LIN {X 102.988,Y 84.879,Z 70.201,A 180.000,B 0.000,C 180.000} C_DIS
LIN {X 102.919,Y 84.847,Z 70.198,A 180.000,B 0.000,C 180.000} C_DIS
LIN {X 102.851,Y 84.815,Z 70.196,A 180.000,B 0.000,C 180.000} C_DIS
LIN {X 102.783,Y 84.784,Z 70.193,A 180.000,B 0.000,C 180.000} C_DIS
LIN {X 102.714,Y 84.755,Z 70.191,A 180.000,B 0.000,C 180.000} C_DIS
LIN {X 102.644,Y 84.727,Z 70.188,A 180.000,B 0.000,C 180.000} C_DIS
LIN {X 102.573,Y 84.698,Z 70.185,A 180.000,B 0.000,C 180.000} C_DIS
LIN {X 102.502,Y 84.670,Z 70.183,A 180.000,B 0.000,C 180.000} C_DIS
LIN {X 102.432,Y 84.642,Z 70.180,A 180.000,B 0.000,C 180.000} C_DIS
LIN {X 102.361,Y 84.613,Z 70.177,A 180.000,B 0.000,C 180.000} C_DIS
LIN {X 102.290,Y 84.585,Z 70.175,A 180.000,B 0.000,C 180.000} C_DIS
LIN {X 102.220,Y 84.557,Z 70.172,A 180.000,B 0.000,C 180.000} C_DIS
LIN {X 102.149,Y 84.528,Z 70.169,A 180.000,B 0.000,C 180.000} C_DIS
LIN {X 102.078,Y 84.501,Z 70.167,A 180.000,B 0.000,C 180.000} C_DIS
LIN {X 102.007,Y 84.475,Z 70.164,A 180.000,B 0.000,C 180.000} C_DIS
LIN {X 101.936,Y 84.451,Z 70.161,A 180.000,B 0.000,C 180.000} C_DIS
LIN {X 101.864,Y 84.427,Z 70.159,A 180.000,B 0.000,C 180.000} C_DIS
LIN {X 101.793,Y 84.403,Z 70.156,A 180.000,B 0.000,C 180.000} C_DIS
LIN {X 101.648,Y 84.354,Z 70.151,A 180.000,B 0.000,C 180.000} C_DIS
LIN {X 101.432,Y 84.281,Z 70.143,A 180.000,B 0.000,C 180.000} C_DIS
LIN {X 101.360,Y 84.257,Z 70.140,A 180.000,B 0.000,C 180.000} C_DIS
LIN {X 101.288,Y 84.235,Z 70.137,A 180.000,B 0.000,C 180.000} C_DIS
LIN {X 101.215,Y 84.214,Z 70.135,A 180.000,B 0.000,C 180.000} C_DIS
LIN {X 100.995,Y 84.154,Z 70.127,A 180.000,B 0.000,C 180.000} C_DIS
LIN {X 100.702,Y 84.073,Z 70.116,A 180.000,B 0.000,C 180.000} C_DIS
LIN {X 100.629,Y 84.053,Z 70.114,A 180.000,B 0.000,C 180.000} C_DIS
LIN {X 100.555,Y 84.034,Z 70.111,A 180.000,B 0.000,C 180.000} C_DIS
LIN {X 100.481,Y 84.018,Z 70.108,A 180.000,B 0.000,C 180.000} C_DIS
LIN {X 100.258,Y 83.970,Z 70.100,A 180.000,B 0.000,C 180.000} C_DIS
LIN {X 100.109,Y 83.938,Z 70.095,A 180.000,B 0.000,C 180.000} C_DIS
LIN {X 100.034,Y 83.921,Z 70.092,A 180.000,B 0.000,C 180.000} C_DIS
LIN {X 99.960,Y 83.905,Z 70.090,A 180.000,B 0.000,C 180.000} C_DIS
LIN {X 99.886,Y 83.890,Z 70.087,A 180.000,B 0.000,C 180.000} C_DIS
LIN {X 99.812,Y 83.874,Z 70.084,A 180.000,B 0.000,C 180.000} C_DIS
LIN {X 99.737,Y 83.861,Z 70.082,A 180.000,B 0.000,C 180.000} C_DIS
LIN {X 99.661,Y 83.849,Z 70.079,A 180.000,B 0.000,C 180.000} C_DIS
LIN {X 99.586,Y 83.838,Z 70.076,A 180.000,B 0.000,C 180.000} C_DIS
LIN {X 99.511,Y 83.826,Z 70.074,A 180.000,B 0.000,C 180.000} C_DIS
LIN {X 99.435,Y 83.814,Z 70.071,A 180.000,B 0.000,C 180.000} C_DIS
LIN {X 99.360,Y 83.802,Z 70.068,A 180.000,B 0.000,C 180.000} C_DIS
LIN {X 99.285,Y 83.790,Z 70.066,A 180.000,B 0.000,C 180.000} C_DIS
LIN {X 99.209,Y 83.778,Z 70.063,A 180.000,B 0.000,C 180.000} C_DIS
LIN {X 99.134,Y 83.766,Z 70.060,A 180.000,B 0.000,C 180.000} C_DIS
LIN {X 99.059,Y 83.755,Z 70.058,A 180.000,B 0.000,C 180.000} C_DIS
LIN {X 98.983,Y 83.746,Z 70.055,A 180.000,B 0.000,C 180.000} C_DIS
LIN {X 98.908,Y 83.739,Z 70.052,A 180.000,B 0.000,C 180.000} C_DIS
LIN {X 98.832,Y 83.731,Z 70.050,A 180.000,B 0.000,C 180.000} C_DIS
LIN {X 98.756,Y 83.724,Z 70.047,A 180.000,B 0.000,C 180.000} C_DIS
LIN {X 98.680,Y 83.716,Z 70.044,A 180.000,B 0.000,C 180.000} C_DIS
LIN {X 98.604,Y 83.708,Z 70.042,A 180.000,B 0.000,C 180.000} C_DIS
LIN {X 98.528,Y 83.701,Z 70.039,A 180.000,B 0.000,C 180.000} C_DIS
LIN {X 98.377,Y 83.686,Z 70.035,A 180.000,B 0.000,C 180.000} C_DIS
LIN {X 98.225,Y 83.674,Z 70.030,A 180.000,B 0.000,C 180.000} C_DIS
LIN {X 98.073,Y 83.667,Z 70.026,A 180.000,B 0.000,C 180.000} C_DIS
LIN {X 97.920,Y 83.661,Z 70.021,A 180.000,B 0.000,C 180.000} C_DIS
LIN {X 97.768,Y 83.655,Z 70.018,A 180.000,B 0.000,C 180.000} C_DIS
LIN {X 97.615,Y 83.649,Z 70.014,A 180.000,B 0.000,C 180.000} C_DIS
LIN {X 97.463,Y 83.646,Z 70.011,A 180.000,B 0.000,C 180.000} C_DIS
LIN {X 97.310,Y 83.648,Z 70.008,A 180.000,B 0.000,C 180.000} C_DIS
LIN {X 97.005,Y 83.655,Z 70.004,A 180.000,B 0.000,C 180.000} C_DIS
LIN {X 96.700,Y 83.664,Z 70.001,A 180.000,B 0.000,C 180.000} C_DIS
LIN {X 96.396,Y 83.689,Z 70.000,A 180.000,B 0.000,C 180.000} C_DIS
LIN {X 96.368,Y 83.693,Z 70.000,A 180.000,B 0.000,C 180.000} C_DIS
; Cutting Move Starts
LIN {X 96.181,Y 83.709,Z 70.000,A 180.000,B 0.000,C 180.000} C_DIS
LIN {X 96.003,Y 83.724,Z 70.000,A 180.000,B 0.000,C 180.000} C_DIS
LIN {X 95.824,Y 83.746,Z 70.000,A 180.000,B 0.000,C 180.000} C_DIS
LIN {X 95.288,Y 83.822,Z 70.000,A 180.000,B 0.000,C 180.000} C_DIS
LIN {X 95.137,Y 83.846,Z 70.000,A 180.000,B 0.000,C 180.000} C_DIS
LIN {X 95.109,Y 83.852,Z 70.000,A 180.000,B 0.000,C 180.000} C_DIS
LIN {X 94.930,Y 83.887,Z 70.000,A 180.000,B 0.000,C 180.000} C_DIS
LIN {X 94.573,Y 83.958,Z 70.000,A 180.000,B 0.000,C 180.000} C_DIS
LIN {X 94.394,Y 83.995,Z 70.000,A 180.000,B 0.000,C 180.000} C_DIS
LIN {X 94.276,Y 84.025,Z 70.000,A 180.000,B 0.000,C 180.000} C_DIS
LIN {X 93.857,Y 84.133,Z 70.000,A 180.000,B 0.000,C 180.000} C_DIS
LIN {X 93.679,Y 84.180,Z 70.000,A 180.000,B 0.000,C 180.000} C_DIS
LIN {X 93.600,Y 84.204,Z 70.000,A 180.000,B 0.000,C 180.000} C_DIS
LIN {X 93.039,Y 84.383,Z 70.000,A 180.000,B 0.000,C 180.000} C_DIS
LIN {X 92.964,Y 84.407,Z 70.000,A 180.000,B 0.000,C 180.000} C_DIS
LIN {X 92.785,Y 84.472,Z 70.000,A 180.000,B 0.000,C 180.000} C_DIS
LIN {X 92.427,Y 84.608,Z 70.000,A 180.000,B 0.000,C 180.000} C_DIS
LIN {X 92.249,Y 84.677,Z 70.000,A 180.000,B 0.000,C 180.000} C_DIS
LIN {X 92.099,Y 84.740,Z 70.000,A 180.000,B 0.000,C 180.000} C_DIS
LIN {X 91.700,Y 84.919,Z 70.000,A 180.000,B 0.000,C 180.000} C_DIS
LIN {X 91.533,Y 84.994,Z 70.000,A 180.000,B 0.000,C 180.000} C_DIS
LIN {X 91.355,Y 85.082,Z 70.000,A 180.000,B 0.000,C 180.000} C_DIS
LIN {X 90.979,Y 85.276,Z 70.000,A 180.000,B 0.000,C 180.000} C_DIS
LIN {X 90.818,Y 85.360,Z 70.000,A 180.000,B 0.000,C 180.000} C_DIS
LIN {X 90.653,Y 85.455,Z 70.000,A 180.000,B 0.000,C 180.000} C_DIS
LIN {X 90.282,Y 85.674,Z 70.000,A 180.000,B 0.000,C 180.000} C_DIS
LIN {X 90.103,Y 85.782,Z 70.000,A 180.000,B 0.000,C 180.000} C_DIS
LIN {X 90.057,Y 85.813,Z 70.000,A 180.000,B 0.000,C 180.000} C_DIS
LIN {X 89.567,Y 86.140,Z 70.000,A 180.000,B 0.000,C 180.000} C_DIS
LIN {X 89.522,Y 86.170,Z 70.000,A 180.000,B 0.000,C 180.000} C_DIS
LIN {X 89.388,Y 86.267,Z 70.000,A 180.000,B 0.000,C 180.000} C_DIS
LIN {X 89.031,Y 86.536,Z 70.000,A 180.000,B 0.000,C 180.000} C_DIS
LIN {X 88.852,Y 86.673,Z 70.000,A 180.000,B 0.000,C 180.000} C_DIS
LIN {X 88.811,Y 86.707,Z 70.000,A 180.000,B 0.000,C 180.000} C_DIS
LIN {X 88.673,Y 86.823,Z 70.000,A 180.000,B 0.000,C 180.000} C_DIS
LIN {X 88.316,Y 87.125,Z 70.000,A 180.000,B 0.000,C 180.000} C_DIS
LIN {X 88.184,Y 87.243,Z 70.000,A 180.000,B 0.000,C 180.000} C_DIS
LIN {X 87.779,Y 87.626,Z 70.000,A 180.000,B 0.000,C 180.000} C_DIS
LIN {X 87.627,Y 87.779,Z 70.000,A 180.000,B 0.000,C 180.000} C_DIS
LIN {X 87.243,Y 88.185,Z 70.000,A 180.000,B 0.000,C 180.000} C_DIS
LIN {X 87.124,Y 88.316,Z 70.000,A 180.000,B 0.000,C 180.000} C_DIS
LIN {X 87.064,Y 88.386,Z 70.000,A 180.000,B 0.000,C 180.000} C_DIS
LIN {X 86.822,Y 88.673,Z 70.000,A 180.000,B 0.000,C 180.000} C_DIS
LIN {X 86.707,Y 88.810,Z 70.000,A 180.000,B 0.000,C 180.000} C_DIS
LIN {X 86.672,Y 88.852,Z 70.000,A 180.000,B 0.000,C 180.000} C_DIS
LIN {X 86.536,Y 89.031,Z 70.000,A 180.000,B 0.000,C 180.000} C_DIS
LIN {X 86.267,Y 89.388,Z 70.000,A 180.000,B 0.000,C 180.000} C_DIS
LIN {X 86.170,Y 89.522,Z 70.000,A 180.000,B 0.000,C 180.000} C_DIS
LIN {X 86.140,Y 89.567,Z 70.000,A 180.000,B 0.000,C 180.000} C_DIS
LIN {X 85.813,Y 90.056,Z 70.000,A 180.000,B 0.000,C 180.000} C_DIS
LIN {X 85.782,Y 90.103,Z 70.000,A 180.000,B 0.000,C 180.000} C_DIS
LIN {X 85.674,Y 90.282,Z 70.000,A 180.000,B 0.000,C 180.000} C_DIS
LIN {X 85.455,Y 90.653,Z 70.000,A 180.000,B 0.000,C 180.000} C_DIS
LIN {X 85.360,Y 90.818,Z 70.000,A 180.000,B 0.000,C 180.000} C_DIS
LIN {X 85.276,Y 90.979,Z 70.000,A 180.000,B 0.000,C 180.000} C_DIS
LIN {X 85.082,Y 91.355,Z 70.000,A 180.000,B 0.000,C 180.000} C_DIS
LIN {X 84.993,Y 91.533,Z 70.000,A 180.000,B 0.000,C 180.000} C_DIS
LIN {X 84.919,Y 91.699,Z 70.000,A 180.000,B 0.000,C 180.000} C_DIS
LIN {X 84.740,Y 92.099,Z 70.000,A 180.000,B 0.000,C 180.000} C_DIS
LIN {X 84.677,Y 92.249,Z 70.000,A 180.000,B 0.000,C 180.000} C_DIS
LIN {X 84.609,Y 92.427,Z 70.000,A 180.000,B 0.000,C 180.000} C_DIS
LIN {X 84.472,Y 92.785,Z 70.000,A 180.000,B 0.000,C 180.000} C_DIS
LIN {X 84.406,Y 92.964,Z 70.000,A 180.000,B 0.000,C 180.000} C_DIS
LIN {X 84.383,Y 93.037,Z 70.000,A 180.000,B 0.000,C 180.000} C_DIS
LIN {X 84.235,Y 93.500,Z 70.000,A 180.000,B 0.000,C 180.000} C_DIS
LIN {X 84.204,Y 93.598,Z 70.000,A 180.000,B 0.000,C 180.000} C_DIS
LIN {X 84.180,Y 93.679,Z 70.000,A 180.000,B 0.000,C 180.000} C_DIS
LIN {X 84.134,Y 93.857,Z 70.000,A 180.000,B 0.000,C 180.000} C_DIS
LIN {X 84.025,Y 94.278,Z 70.000,A 180.000,B 0.000,C 180.000} C_DIS
LIN {X 83.996,Y 94.394,Z 70.000,A 180.000,B 0.000,C 180.000} C_DIS
LIN {X 83.958,Y 94.573,Z 70.000,A 180.000,B 0.000,C 180.000} C_DIS
LIN {X 83.851,Y 95.109,Z 70.000,A 180.000,B 0.000,C 180.000} C_DIS
LIN {X 83.846,Y 95.134,Z 70.000,A 180.000,B 0.000,C 180.000} C_DIS
LIN {X 83.822,Y 95.288,Z 70.000,A 180.000,B 0.000,C 180.000} C_DIS
LIN {X 83.746,Y 95.824,Z 70.000,A 180.000,B 0.000,C 180.000} C_DIS
LIN {X 83.724,Y 96.003,Z 70.000,A 180.000,B 0.000,C 180.000} C_DIS
LIN {X 83.709,Y 96.181,Z 70.000,A 180.000,B 0.000,C 180.000} C_DIS
LIN {X 83.679,Y 96.539,Z 70.000,A 180.000,B 0.000,C 180.000} C_DIS
LIN {X 83.668,Y 96.673,Z 70.000,A 180.000,B 0.000,C 180.000} C_DIS
LIN {X 83.665,Y 96.718,Z 70.000,A 180.000,B 0.000,C 180.000} C_DIS
LIN {X 83.659,Y 96.897,Z 70.000,A 180.000,B 0.000,C 180.000} C_DIS
LIN {X 83.648,Y 97.254,Z 70.000,A 180.000,B 0.000,C 180.000} C_DIS
LIN {X 83.644,Y 97.433,Z 70.000,A 180.000,B 0.000,C 180.000} C_DIS
LIN {X 83.645,Y 97.612,Z 70.000,A 180.000,B 0.000,C 180.000} C_DIS
LIN {X 83.660,Y 98.148,Z 70.000,A 180.000,B 0.000,C 180.000} C_DIS
LIN {X 83.668,Y 98.327,Z 70.000,A 180.000,B 0.000,C 180.000} C_DIS
LIN {X 83.683,Y 98.505,Z 70.000,A 180.000,B 0.000,C 180.000} C_DIS
LIN {X 83.713,Y 98.863,Z 70.000,A 180.000,B 0.000,C 180.000} C_DIS
LIN {X 83.729,Y 99.042,Z 70.000,A 180.000,B 0.000,C 180.000} C_DIS
LIN {X 83.753,Y 99.221,Z 70.000,A 180.000,B 0.000,C 180.000} C_DIS
LIN {X 83.828,Y 99.757,Z 70.000,A 180.000,B 0.000,C 180.000} C_DIS
LIN {X 83.846,Y 99.866,Z 70.000,A 180.000,B 0.000,C 180.000} C_DIS
LIN {X 83.860,Y 99.936,Z 70.000,A 180.000,B 0.000,C 180.000} C_DIS
LIN {X 83.967,Y 100.472,Z 70.000,A 180.000,B 0.000,C 180.000} C_DIS
LIN {X 84.007,Y 100.651,Z 70.000,A 180.000,B 0.000,C 180.000} C_DIS
LIN {X 84.025,Y 100.722,Z 70.000,A 180.000,B 0.000,C 180.000} C_DIS
LIN {X 84.145,Y 101.187,Z 70.000,A 180.000,B 0.000,C 180.000} C_DIS
LIN {X 84.193,Y 101.366,Z 70.000,A 180.000,B 0.000,C 180.000} C_DIS
LIN {X 84.204,Y 101.402,Z 70.000,A 180.000,B 0.000,C 180.000} C_DIS
LIN {X 84.249,Y 101.545,Z 70.000,A 180.000,B 0.000,C 180.000} C_DIS
LIN {X 84.383,Y 101.963,Z 70.000,A 180.000,B 0.000,C 180.000} C_DIS
LIN {X 84.422,Y 102.081,Z 70.000,A 180.000,B 0.000,C 180.000} C_DIS
LIN {X 84.489,Y 102.260,Z 70.000,A 180.000,B 0.000,C 180.000} C_DIS
LIN {X 84.626,Y 102.617,Z 70.000,A 180.000,B 0.000,C 180.000} C_DIS
LIN {X 84.695,Y 102.796,Z 70.000,A 180.000,B 0.000,C 180.000} C_DIS
LIN {X 84.740,Y 102.901,Z 70.000,A 180.000,B 0.000,C 180.000} C_DIS
LIN {X 84.933,Y 103.332,Z 70.000,A 180.000,B 0.000,C 180.000} C_DIS
LIN {X 85.014,Y 103.511,Z 70.000,A 180.000,B 0.000,C 180.000} C_DIS
LIN {X 85.098,Y 103.675,Z 70.000,A 180.000,B 0.000,C 180.000} C_DIS
LIN {X 85.290,Y 104.047,Z 70.000,A 180.000,B 0.000,C 180.000} C_DIS
LIN {X 85.385,Y 104.226,Z 70.000,A 180.000,B 0.000,C 180.000} C_DIS
LIN {X 85.455,Y 104.347,Z 70.000,A 180.000,B 0.000,C 180.000} C_DIS
LIN {X 85.700,Y 104.762,Z 70.000,A 180.000,B 0.000,C 180.000} C_DIS
LIN {X 85.811,Y 104.941,Z 70.000,A 180.000,B 0.000,C 180.000} C_DIS
LIN {X 86.050,Y 105.299,Z 70.000,A 180.000,B 0.000,C 180.000} C_DIS
LIN {X 86.170,Y 105.477,Z 70.000,A 180.000,B 0.000,C 180.000} C_DIS
LIN {X 86.170,Y 105.478,Z 70.000,A 180.000,B 0.000,C 180.000} C_DIS
LIN {X 86.301,Y 105.656,Z 70.000,A 180.000,B 0.000,C 180.000} C_DIS
LIN {X 86.570,Y 106.014,Z 70.000,A 180.000,B 0.000,C 180.000} C_DIS
LIN {X 86.707,Y 106.190,Z 70.000,A 180.000,B 0.000,C 180.000} C_DIS
LIN {X 86.709,Y 106.193,Z 70.000,A 180.000,B 0.000,C 180.000} C_DIS
LIN {X 86.885,Y 106.402,Z 70.000,A 180.000,B 0.000,C 180.000} C_DIS
LIN {X 87.064,Y 106.614,Z 70.000,A 180.000,B 0.000,C 180.000} C_DIS
LIN {X 87.163,Y 106.729,Z 70.000,A 180.000,B 0.000,C 180.000} C_DIS
LIN {X 87.243,Y 106.815,Z 70.000,A 180.000,B 0.000,C 180.000} C_DIS
LIN {X 87.601,Y 107.193,Z 70.000,A 180.000,B 0.000,C 180.000} C_DIS
LIN {X 87.669,Y 107.265,Z 70.000,A 180.000,B 0.000,C 180.000} C_DIS
LIN {X 87.779,Y 107.374,Z 70.000,A 180.000,B 0.000,C 180.000} C_DIS
LIN {X 88.137,Y 107.712,Z 70.000,A 180.000,B 0.000,C 180.000} C_DIS
LIN {X 88.232,Y 107.802,Z 70.000,A 180.000,B 0.000,C 180.000} C_DIS
LIN {X 88.316,Y 107.875,Z 70.000,A 180.000,B 0.000,C 180.000} C_DIS
LIN {X 88.673,Y 108.177,Z 70.000,A 180.000,B 0.000,C 180.000} C_DIS
LIN {X 88.852,Y 108.327,Z 70.000,A 180.000,B 0.000,C 180.000} C_DIS
LIN {X 88.865,Y 108.338,Z 70.000,A 180.000,B 0.000,C 180.000} C_DIS
LIN {X 89.031,Y 108.464,Z 70.000,A 180.000,B 0.000,C 180.000} C_DIS
LIN {X 89.388,Y 108.733,Z 70.000,A 180.000,B 0.000,C 180.000} C_DIS
LIN {X 89.567,Y 108.860,Z 70.000,A 180.000,B 0.000,C 180.000} C_DIS
LIN {X 89.925,Y 109.099,Z 70.000,A 180.000,B 0.000,C 180.000} C_DIS
LIN {X 90.103,Y 109.218,Z 70.000,A 180.000,B 0.000,C 180.000} C_DIS
LIN {X 90.125,Y 109.232,Z 70.000,A 180.000,B 0.000,C 180.000} C_DIS
LIN {X 90.282,Y 109.326,Z 70.000,A 180.000,B 0.000,C 180.000} C_DIS
LIN {X 90.728,Y 109.589,Z 70.000,A 180.000,B 0.000,C 180.000} C_DIS
LIN {X 90.818,Y 109.640,Z 70.000,A 180.000,B 0.000,C 180.000} C_DIS
LIN {X 90.997,Y 109.733,Z 70.000,A 180.000,B 0.000,C 180.000} C_DIS
LIN {X 91.411,Y 109.947,Z 70.000,A 180.000,B 0.000,C 180.000} C_DIS
LIN {X 91.533,Y 110.006,Z 70.000,A 180.000,B 0.000,C 180.000} C_DIS
LIN {X 91.712,Y 110.087,Z 70.000,A 180.000,B 0.000,C 180.000} C_DIS
LIN {X 92.070,Y 110.247,Z 70.000,A 180.000,B 0.000,C 180.000} C_DIS
LIN {X 92.201,Y 110.304,Z 70.000,A 180.000,B 0.000,C 180.000} C_DIS
LIN {X 92.249,Y 110.323,Z 70.000,A 180.000,B 0.000,C 180.000} C_DIS
LIN {X 92.427,Y 110.392,Z 70.000,A 180.000,B 0.000,C 180.000} C_DIS
LIN {X 92.785,Y 110.528,Z 70.000,A 180.000,B 0.000,C 180.000} C_DIS
LIN {X 92.964,Y 110.593,Z 70.000,A 180.000,B 0.000,C 180.000} C_DIS
LIN {X 93.142,Y 110.650,Z 70.000,A 180.000,B 0.000,C 180.000} C_DIS
LIN {X 93.500,Y 110.764,Z 70.000,A 180.000,B 0.000,C 180.000} C_DIS
LIN {X 93.679,Y 110.820,Z 70.000,A 180.000,B 0.000,C 180.000} C_DIS
LIN {X 93.755,Y 110.841,Z 70.000,A 180.000,B 0.000,C 180.000} C_DIS
LIN {X 94.215,Y 110.959,Z 70.000,A 180.000,B 0.000,C 180.000} C_DIS
LIN {X 94.394,Y 111.005,Z 70.000,A 180.000,B 0.000,C 180.000} C_DIS
LIN {X 94.460,Y 111.019,Z 70.000,A 180.000,B 0.000,C 180.000} C_DIS
LIN {X 94.573,Y 111.042,Z 70.000,A 180.000,B 0.000,C 180.000} C_DIS
LIN {X 94.930,Y 111.113,Z 70.000,A 180.000,B 0.000,C 180.000} C_DIS
LIN {X 95.109,Y 111.148,Z 70.000,A 180.000,B 0.000,C 180.000} C_DIS
LIN {X 95.288,Y 111.178,Z 70.000,A 180.000,B 0.000,C 180.000} C_DIS
LIN {X 95.824,Y 111.254,Z 70.000,A 180.000,B 0.000,C 180.000} C_DIS
LIN {X 96.003,Y 111.276,Z 70.000,A 180.000,B 0.000,C 180.000} C_DIS
LIN {X 96.181,Y 111.291,Z 70.000,A 180.000,B 0.000,C 180.000} C_DIS
LIN {X 96.539,Y 111.321,Z 70.000,A 180.000,B 0.000,C 180.000} C_DIS
LIN {X 96.718,Y 111.335,Z 70.000,A 180.000,B 0.000,C 180.000} C_DIS
LIN {X 96.897,Y 111.342,Z 70.000,A 180.000,B 0.000,C 180.000} C_DIS
LIN {X 97.433,Y 111.357,Z 70.000,A 180.000,B 0.000,C 180.000} C_DIS
LIN {X 97.612,Y 111.355,Z 70.000,A 180.000,B 0.000,C 180.000} C_DIS
LIN {X 98.148,Y 111.340,Z 70.000,A 180.000,B 0.000,C 180.000} C_DIS
LIN {X 98.327,Y 111.332,Z 70.000,A 180.000,B 0.000,C 180.000} C_DIS
LIN {X 98.505,Y 111.317,Z 70.000,A 180.000,B 0.000,C 180.000} C_DIS
LIN {X 98.863,Y 111.287,Z 70.000,A 180.000,B 0.000,C 180.000} C_DIS
LIN {X 99.042,Y 111.271,Z 70.000,A 180.000,B 0.000,C 180.000} C_DIS
LIN {X 99.221,Y 111.248,Z 70.000,A 180.000,B 0.000,C 180.000} C_DIS
LIN {X 99.578,Y 111.197,Z 70.000,A 180.000,B 0.000,C 180.000} C_DIS
LIN {X 99.757,Y 111.172,Z 70.000,A 180.000,B 0.000,C 180.000} C_DIS
LIN {X 99.936,Y 111.140,Z 70.000,A 180.000,B 0.000,C 180.000} C_DIS
LIN {X 100.472,Y 111.033,Z 70.000,A 180.000,B 0.000,C 180.000} C_DIS
LIN {X 100.540,Y 111.019,Z 70.000,A 180.000,B 0.000,C 180.000} C_DIS
LIN {X 100.651,Y 110.994,Z 70.000,A 180.000,B 0.000,C 180.000} C_DIS
LIN {X 100.829,Y 110.948,Z 70.000,A 180.000,B 0.000,C 180.000} C_DIS
LIN {X 101.245,Y 110.841,Z 70.000,A 180.000,B 0.000,C 180.000} C_DIS
LIN {X 101.366,Y 110.807,Z 70.000,A 180.000,B 0.000,C 180.000} C_DIS
LIN {X 101.545,Y 110.750,Z 70.000,A 180.000,B 0.000,C 180.000} C_DIS
LIN {X 101.902,Y 110.636,Z 70.000,A 180.000,B 0.000,C 180.000} C_DIS
LIN {X 102.081,Y 110.578,Z 70.000,A 180.000,B 0.000,C 180.000} C_DIS
LIN {X 102.260,Y 110.511,Z 70.000,A 180.000,B 0.000,C 180.000} C_DIS
LIN {X 102.617,Y 110.375,Z 70.000,A 180.000,B 0.000,C 180.000} C_DIS
LIN {X 102.796,Y 110.306,Z 70.000,A 180.000,B 0.000,C 180.000} C_DIS
LIN {X 102.799,Y 110.304,Z 70.000,A 180.000,B 0.000,C 180.000} C_DIS
LIN {X 102.975,Y 110.227,Z 70.000,A 180.000,B 0.000,C 180.000} C_DIS
LIN {X 103.332,Y 110.067,Z 70.000,A 180.000,B 0.000,C 180.000} C_DIS
LIN {X 103.511,Y 109.985,Z 70.000,A 180.000,B 0.000,C 180.000} C_DIS
LIN {X 103.589,Y 109.947,Z 70.000,A 180.000,B 0.000,C 180.000} C_DIS
LIN {X 104.047,Y 109.710,Z 70.000,A 180.000,B 0.000,C 180.000} C_DIS
LIN {X 104.226,Y 109.616,Z 70.000,A 180.000,B 0.000,C 180.000} C_DIS
LIN {X 104.272,Y 109.589,Z 70.000,A 180.000,B 0.000,C 180.000} C_DIS
LIN {X 104.762,Y 109.300,Z 70.000,A 180.000,B 0.000,C 180.000} C_DIS
LIN {X 104.875,Y 109.232,Z 70.000,A 180.000,B 0.000,C 180.000} C_DIS
LIN {X 104.941,Y 109.189,Z 70.000,A 180.000,B 0.000,C 180.000} C_DIS
LIN {X 105.145,Y 109.053,Z 70.000,A 180.000,B 0.000,C 180.000} C_DIS
LIN {X 105.412,Y 108.874,Z 70.000,A 180.000,B 0.000,C 180.000} C_DIS
LIN {X 105.477,Y 108.830,Z 70.000,A 180.000,B 0.000,C 180.000} C_DIS
LIN {X 105.656,Y 108.700,Z 70.000,A 180.000,B 0.000,C 180.000} C_DIS
LIN {X 106.014,Y 108.431,Z 70.000,A 180.000,B 0.000,C 180.000} C_DIS
LIN {X 106.135,Y 108.338,Z 70.000,A 180.000,B 0.000,C 180.000} C_DIS
LIN {X 106.193,Y 108.291,Z 70.000,A 180.000,B 0.000,C 180.000} C_DIS
LIN {X 106.349,Y 108.159,Z 70.000,A 180.000,B 0.000,C 180.000} C_DIS
LIN {X 106.560,Y 107.980,Z 70.000,A 180.000,B 0.000,C 180.000} C_DIS
LIN {X 106.729,Y 107.837,Z 70.000,A 180.000,B 0.000,C 180.000} C_DIS
LIN {X 106.768,Y 107.802,Z 70.000,A 180.000,B 0.000,C 180.000} C_DIS
LIN {X 106.908,Y 107.670,Z 70.000,A 180.000,B 0.000,C 180.000} C_DIS
LIN {X 107.147,Y 107.444,Z 70.000,A 180.000,B 0.000,C 180.000} C_DIS
LIN {X 107.265,Y 107.332,Z 70.000,A 180.000,B 0.000,C 180.000} C_DIS
LIN {X 107.331,Y 107.265,Z 70.000,A 180.000,B 0.000,C 180.000} C_DIS
LIN {X 107.444,Y 107.146,Z 70.000,A 180.000,B 0.000,C 180.000} C_DIS
LIN {X 107.669,Y 106.908,Z 70.000,A 180.000,B 0.000,C 180.000} C_DIS
LIN {X 107.802,Y 106.768,Z 70.000,A 180.000,B 0.000,C 180.000} C_DIS
LIN {X 107.837,Y 106.729,Z 70.000,A 180.000,B 0.000,C 180.000} C_DIS
LIN {X 107.980,Y 106.561,Z 70.000,A 180.000,B 0.000,C 180.000} C_DIS
LIN {X 108.159,Y 106.349,Z 70.000,A 180.000,B 0.000,C 180.000} C_DIS
LIN {X 108.291,Y 106.193,Z 70.000,A 180.000,B 0.000,C 180.000} C_DIS
LIN {X 108.338,Y 106.135,Z 70.000,A 180.000,B 0.000,C 180.000} C_DIS
LIN {X 108.430,Y 106.014,Z 70.000,A 180.000,B 0.000,C 180.000} C_DIS
LIN {X 108.699,Y 105.656,Z 70.000,A 180.000,B 0.000,C 180.000} C_DIS
LIN {X 108.830,Y 105.477,Z 70.000,A 180.000,B 0.000,C 180.000} C_DIS
LIN {X 108.874,Y 105.412,Z 70.000,A 180.000,B 0.000,C 180.000} C_DIS
LIN {X 109.189,Y 104.941,Z 70.000,A 180.000,B 0.000,C 180.000} C_DIS
LIN {X 109.232,Y 104.876,Z 70.000,A 180.000,B 0.000,C 180.000} C_DIS
LIN {X 109.300,Y 104.762,Z 70.000,A 180.000,B 0.000,C 180.000} C_DIS
LIN {X 109.511,Y 104.405,Z 70.000,A 180.000,B 0.000,C 180.000} C_DIS
LIN {X 109.589,Y 104.271,Z 70.000,A 180.000,B 0.000,C 180.000} C_DIS
LIN {X 109.615,Y 104.226,Z 70.000,A 180.000,B 0.000,C 180.000} C_DIS
LIN {X 109.710,Y 104.047,Z 70.000,A 180.000,B 0.000,C 180.000} C_DIS
LIN {X 109.947,Y 103.589,Z 70.000,A 180.000,B 0.000,C 180.000} C_DIS
LIN {X 109.986,Y 103.511,Z 70.000,A 180.000,B 0.000,C 180.000} C_DIS
LIN {X 110.067,Y 103.332,Z 70.000,A 180.000,B 0.000,C 180.000} C_DIS
LIN {X 110.227,Y 102.975,Z 70.000,A 180.000,B 0.000,C 180.000} C_DIS
LIN {X 110.304,Y 102.798,Z 70.000,A 180.000,B 0.000,C 180.000} C_DIS
LIN {X 110.305,Y 102.796,Z 70.000,A 180.000,B 0.000,C 180.000} C_DIS
LIN {X 110.374,Y 102.617,Z 70.000,A 180.000,B 0.000,C 180.000} C_DIS
LIN {X 110.511,Y 102.260,Z 70.000,A 180.000,B 0.000,C 180.000} C_DIS
LIN {X 110.578,Y 102.081,Z 70.000,A 180.000,B 0.000,C 180.000} C_DIS
LIN {X 110.637,Y 101.902,Z 70.000,A 180.000,B 0.000,C 180.000} C_DIS
LIN {X 110.751,Y 101.545,Z 70.000,A 180.000,B 0.000,C 180.000} C_DIS
LIN {X 110.807,Y 101.366,Z 70.000,A 180.000,B 0.000,C 180.000} C_DIS
LIN {X 110.841,Y 101.243,Z 70.000,A 180.000,B 0.000,C 180.000} C_DIS
LIN {X 110.947,Y 100.829,Z 70.000,A 180.000,B 0.000,C 180.000} C_DIS
LIN {X 110.993,Y 100.651,Z 70.000,A 180.000,B 0.000,C 180.000} C_DIS
LIN {X 111.019,Y 100.541,Z 70.000,A 180.000,B 0.000,C 180.000} C_DIS
LIN {X 111.033,Y 100.472,Z 70.000,A 180.000,B 0.000,C 180.000} C_DIS
LIN {X 111.140,Y 99.936,Z 70.000,A 180.000,B 0.000,C 180.000} C_DIS
LIN {X 111.172,Y 99.757,Z 70.000,A 180.000,B 0.000,C 180.000} C_DIS
LIN {X 111.247,Y 99.221,Z 70.000,A 180.000,B 0.000,C 180.000} C_DIS
LIN {X 111.271,Y 99.042,Z 70.000,A 180.000,B 0.000,C 180.000} C_DIS
LIN {X 111.287,Y 98.863,Z 70.000,A 180.000,B 0.000,C 180.000} C_DIS
LIN {X 111.317,Y 98.505,Z 70.000,A 180.000,B 0.000,C 180.000} C_DIS
LIN {X 111.332,Y 98.327,Z 70.000,A 180.000,B 0.000,C 180.000} C_DIS
LIN {X 111.340,Y 98.148,Z 70.000,A 180.000,B 0.000,C 180.000} C_DIS
LIN {X 111.355,Y 97.612,Z 70.000,A 180.000,B 0.000,C 180.000} C_DIS
LIN {X 111.356,Y 97.433,Z 70.000,A 180.000,B 0.000,C 180.000} C_DIS
LIN {X 111.352,Y 97.254,Z 70.000,A 180.000,B 0.000,C 180.000} C_DIS
LIN {X 111.341,Y 96.897,Z 70.000,A 180.000,B 0.000,C 180.000} C_DIS
LIN {X 111.335,Y 96.718,Z 70.000,A 180.000,B 0.000,C 180.000} C_DIS
LIN {X 111.321,Y 96.539,Z 70.000,A 180.000,B 0.000,C 180.000} C_DIS
LIN {X 111.291,Y 96.181,Z 70.000,A 180.000,B 0.000,C 180.000} C_DIS
LIN {X 111.276,Y 96.003,Z 70.000,A 180.000,B 0.000,C 180.000} C_DIS
LIN {X 111.254,Y 95.824,Z 70.000,A 180.000,B 0.000,C 180.000} C_DIS
LIN {X 111.178,Y 95.288,Z 70.000,A 180.000,B 0.000,C 180.000} C_DIS
LIN {X 111.149,Y 95.109,Z 70.000,A 180.000,B 0.000,C 180.000} C_DIS
LIN {X 111.042,Y 94.573,Z 70.000,A 180.000,B 0.000,C 180.000} C_DIS
LIN {X 111.019,Y 94.459,Z 70.000,A 180.000,B 0.000,C 180.000} C_DIS
LIN {X 111.004,Y 94.394,Z 70.000,A 180.000,B 0.000,C 180.000} C_DIS
LIN {X 110.959,Y 94.215,Z 70.000,A 180.000,B 0.000,C 180.000} C_DIS
LIN {X 110.841,Y 93.757,Z 70.000,A 180.000,B 0.000,C 180.000} C_DIS
LIN {X 110.820,Y 93.679,Z 70.000,A 180.000,B 0.000,C 180.000} C_DIS
LIN {X 110.765,Y 93.500,Z 70.000,A 180.000,B 0.000,C 180.000} C_DIS
LIN {X 110.651,Y 93.142,Z 70.000,A 180.000,B 0.000,C 180.000} C_DIS
LIN {X 110.594,Y 92.964,Z 70.000,A 180.000,B 0.000,C 180.000} C_DIS
LIN {X 110.528,Y 92.785,Z 70.000,A 180.000,B 0.000,C 180.000} C_DIS
LIN {X 110.391,Y 92.427,Z 70.000,A 180.000,B 0.000,C 180.000} C_DIS
LIN {X 110.323,Y 92.249,Z 70.000,A 180.000,B 0.000,C 180.000} C_DIS
LIN {X 110.304,Y 92.202,Z 70.000,A 180.000,B 0.000,C 180.000} C_DIS
LIN {X 110.247,Y 92.070,Z 70.000,A 180.000,B 0.000,C 180.000} C_DIS
LIN {X 110.087,Y 91.712,Z 70.000,A 180.000,B 0.000,C 180.000} C_DIS
LIN {X 110.007,Y 91.533,Z 70.000,A 180.000,B 0.000,C 180.000} C_DIS
LIN {X 109.947,Y 91.411,Z 70.000,A 180.000,B 0.000,C 180.000} C_DIS
LIN {X 109.733,Y 90.997,Z 70.000,A 180.000,B 0.000,C 180.000} C_DIS
LIN {X 109.640,Y 90.818,Z 70.000,A 180.000,B 0.000,C 180.000} C_DIS
LIN {X 109.589,Y 90.729,Z 70.000,A 180.000,B 0.000,C 180.000} C_DIS
LIN {X 109.537,Y 90.640,Z 70.000,A 180.000,B 0.000,C 180.000} C_DIS
LIN {X 109.326,Y 90.282,Z 70.000,A 180.000,B 0.000,C 180.000} C_DIS
LIN {X 109.232,Y 90.124,Z 70.000,A 180.000,B 0.000,C 180.000} C_DIS
LIN {X 109.218,Y 90.103,Z 70.000,A 180.000,B 0.000,C 180.000} C_DIS
LIN {X 109.099,Y 89.925,Z 70.000,A 180.000,B 0.000,C 180.000} C_DIS
LIN {X 108.860,Y 89.567,Z 70.000,A 180.000,B 0.000,C 180.000} C_DIS
LIN {X 108.733,Y 89.388,Z 70.000,A 180.000,B 0.000,C 180.000} C_DIS
LIN {X 108.464,Y 89.031,Z 70.000,A 180.000,B 0.000,C 180.000} C_DIS
LIN {X 108.338,Y 88.865,Z 70.000,A 180.000,B 0.000,C 180.000} C_DIS
LIN {X 108.328,Y 88.852,Z 70.000,A 180.000,B 0.000,C 180.000} C_DIS
LIN {X 108.178,Y 88.673,Z 70.000,A 180.000,B 0.000,C 180.000} C_DIS
LIN {X 107.980,Y 88.439,Z 70.000,A 180.000,B 0.000,C 180.000} C_DIS
LIN {X 107.876,Y 88.316,Z 70.000,A 180.000,B 0.000,C 180.000} C_DIS
LIN {X 107.802,Y 88.232,Z 70.000,A 180.000,B 0.000,C 180.000} C_DIS
LIN {X 107.711,Y 88.137,Z 70.000,A 180.000,B 0.000,C 180.000} C_DIS
LIN {X 107.373,Y 87.779,Z 70.000,A 180.000,B 0.000,C 180.000} C_DIS
LIN {X 107.265,Y 87.668,Z 70.000,A 180.000,B 0.000,C 180.000} C_DIS
LIN {X 107.194,Y 87.601,Z 70.000,A 180.000,B 0.000,C 180.000} C_DIS
LIN {X 106.816,Y 87.243,Z 70.000,A 180.000,B 0.000,C 180.000} C_DIS
LIN {X 106.729,Y 87.163,Z 70.000,A 180.000,B 0.000,C 180.000} C_DIS
LIN {X 106.613,Y 87.064,Z 70.000,A 180.000,B 0.000,C 180.000} C_DIS
LIN {X 106.371,Y 86.860,Z 70.000,A 180.000,B 0.000,C 180.000} C_DIS
LIN {X 106.193,Y 86.709,Z 70.000,A 180.000,B 0.000,C 180.000} C_DIS
LIN {X 106.189,Y 86.707,Z 70.000,A 180.000,B 0.000,C 180.000} C_DIS
LIN {X 106.014,Y 86.569,Z 70.000,A 180.000,B 0.000,C 180.000} C_DIS
LIN {X 105.656,Y 86.300,Z 70.000,A 180.000,B 0.000,C 180.000} C_DIS
LIN {X 105.478,Y 86.170,Z 70.000,A 180.000,B 0.000,C 180.000} C_DIS
LIN {X 105.477,Y 86.170,Z 70.000,A 180.000,B 0.000,C 180.000} C_DIS
LIN {X 105.299,Y 86.050,Z 70.000,A 180.000,B 0.000,C 180.000} C_DIS
LIN {X 105.103,Y 85.920,Z 70.000,A 180.000,B 0.000,C 180.000} C_DIS
LIN {X 104.943,Y 85.813,Z 70.000,A 180.000,B 0.000,C 180.000} C_DIS
LIN {X 104.941,Y 85.811,Z 70.000,A 180.000,B 0.000,C 180.000} C_DIS
LIN {X 104.762,Y 85.700,Z 70.000,A 180.000,B 0.000,C 180.000} C_DIS
LIN {X 104.347,Y 85.455,Z 70.000,A 180.000,B 0.000,C 180.000} C_DIS
LIN {X 104.226,Y 85.384,Z 70.000,A 180.000,B 0.000,C 180.000} C_DIS
LIN {X 104.047,Y 85.290,Z 70.000,A 180.000,B 0.000,C 180.000} C_DIS
LIN {X 103.675,Y 85.098,Z 70.000,A 180.000,B 0.000,C 180.000} C_DIS
LIN {X 103.511,Y 85.015,Z 70.000,A 180.000,B 0.000,C 180.000} C_DIS
LIN {X 103.332,Y 84.933,Z 70.000,A 180.000,B 0.000,C 180.000} C_DIS
LIN {X 102.901,Y 84.740,Z 70.000,A 180.000,B 0.000,C 180.000} C_DIS
LIN {X 102.796,Y 84.694,Z 70.000,A 180.000,B 0.000,C 180.000} C_DIS
LIN {X 102.617,Y 84.625,Z 70.000,A 180.000,B 0.000,C 180.000} C_DIS
LIN {X 102.260,Y 84.489,Z 70.000,A 180.000,B 0.000,C 180.000} C_DIS
LIN {X 102.081,Y 84.422,Z 70.000,A 180.000,B 0.000,C 180.000} C_DIS
LIN {X 101.961,Y 84.383,Z 70.000,A 180.000,B 0.000,C 180.000} C_DIS
LIN {X 101.400,Y 84.204,Z 70.000,A 180.000,B 0.000,C 180.000} C_DIS
LIN {X 101.366,Y 84.193,Z 70.000,A 180.000,B 0.000,C 180.000} C_DIS
LIN {X 101.187,Y 84.144,Z 70.000,A 180.000,B 0.000,C 180.000} C_DIS
LIN {X 100.724,Y 84.025,Z 70.000,A 180.000,B 0.000,C 180.000} C_DIS
LIN {X 100.651,Y 84.006,Z 70.000,A 180.000,B 0.000,C 180.000} C_DIS
LIN {X 100.472,Y 83.967,Z 70.000,A 180.000,B 0.000,C 180.000} C_DIS
LIN {X 99.936,Y 83.860,Z 70.000,A 180.000,B 0.000,C 180.000} C_DIS
LIN {X 99.863,Y 83.846,Z 70.000,A 180.000,B 0.000,C 180.000} C_DIS
LIN {X 99.757,Y 83.828,Z 70.000,A 180.000,B 0.000,C 180.000} C_DIS
LIN {X 99.578,Y 83.803,Z 70.000,A 180.000,B 0.000,C 180.000} C_DIS
LIN {X 99.221,Y 83.752,Z 70.000,A 180.000,B 0.000,C 180.000} C_DIS
LIN {X 99.042,Y 83.729,Z 70.000,A 180.000,B 0.000,C 180.000} C_DIS
LIN {X 98.863,Y 83.713,Z 70.000,A 180.000,B 0.000,C 180.000} C_DIS
LIN {X 98.505,Y 83.683,Z 70.000,A 180.000,B 0.000,C 180.000} C_DIS
LIN {X 98.327,Y 83.668,Z 70.000,A 180.000,B 0.000,C 180.000} C_DIS
LIN {X 98.321,Y 83.668,Z 70.000,A 180.000,B 0.000,C 180.000} C_DIS
LIN {X 98.148,Y 83.660,Z 70.000,A 180.000,B 0.000,C 180.000} C_DIS
LIN {X 97.612,Y 83.645,Z 70.000,A 180.000,B 0.000,C 180.000} C_DIS
LIN {X 97.433,Y 83.643,Z 70.000,A 180.000,B 0.000,C 180.000} C_DIS
LIN {X 96.897,Y 83.658,Z 70.000,A 180.000,B 0.000,C 180.000} C_DIS
LIN {X 96.718,Y 83.665,Z 70.000,A 180.000,B 0.000,C 180.000} C_DIS
LIN {X 96.679,Y 83.668,Z 70.000,A 180.000,B 0.000,C 180.000} C_DIS
LIN {X 96.539,Y 83.679,Z 70.000,A 180.000,B 0.000,C 180.000} C_DIS
LIN {X 96.368,Y 83.693,Z 70.000,A 180.000,B 0.000,C 180.000} C_DIS
; Link Move Starts
LIN {X 96.054,Y 83.717,Z 70.000,A 180.000,B 0.000,C 180.000} C_DIS
LIN {X 95.767,Y 83.751,Z 69.999,A 180.000,B 0.000,C 180.000} C_DIS
LIN {X 95.455,Y 83.795,Z 69.998,A 180.000,B 0.000,C 180.000} C_DIS
LIN {X 95.166,Y 83.837,Z 69.996,A 180.000,B 0.000,C 180.000} C_DIS
LIN {X 94.860,Y 83.896,Z 69.994,A 180.000,B 0.000,C 180.000} C_DIS
LIN {X 94.551,Y 83.956,Z 69.992,A 180.000,B 0.000,C 180.000} C_DIS
LIN {X 94.269,Y 84.019,Z 69.989,A 180.000,B 0.000,C 180.000} C_DIS
LIN {X 93.963,Y 84.096,Z 69.986,A 180.000,B 0.000,C 180.000} C_DIS
LIN {X 93.664,Y 84.173,Z 69.982,A 180.000,B 0.000,C 180.000} C_DIS
LIN {X 93.382,Y 84.260,Z 69.978,A 180.000,B 0.000,C 180.000} C_DIS
LIN {X 93.082,Y 84.353,Z 69.974,A 180.000,B 0.000,C 180.000} C_DIS
LIN {X 92.801,Y 84.447,Z 69.969,A 180.000,B 0.000,C 180.000} C_DIS
LIN {X 92.656,Y 84.502,Z 69.966,A 180.000,B 0.000,C 180.000} C_DIS
LIN {X 92.511,Y 84.556,Z 69.964,A 180.000,B 0.000,C 180.000} C_DIS
LIN {X 92.372,Y 84.607,Z 69.961,A 180.000,B 0.000,C 180.000} C_DIS
LIN {X 92.233,Y 84.659,Z 69.958,A 180.000,B 0.000,C 180.000} C_DIS
LIN {X 92.091,Y 84.719,Z 69.955,A 180.000,B 0.000,C 180.000} C_DIS
LIN {X 91.950,Y 84.780,Z 69.952,A 180.000,B 0.000,C 180.000} C_DIS
LIN {X 91.805,Y 84.843,Z 69.949,A 180.000,B 0.000,C 180.000} C_DIS
LIN {X 91.661,Y 84.906,Z 69.946,A 180.000,B 0.000,C 180.000} C_DIS
LIN {X 91.523,Y 84.966,Z 69.943,A 180.000,B 0.000,C 180.000} C_DIS
LIN {X 91.388,Y 85.031,Z 69.939,A 180.000,B 0.000,C 180.000} C_DIS
LIN {X 91.252,Y 85.099,Z 69.936,A 180.000,B 0.000,C 180.000} C_DIS
LIN {X 91.115,Y 85.168,Z 69.932,A 180.000,B 0.000,C 180.000} C_DIS
LIN {X 90.980,Y 85.236,Z 69.929,A 180.000,B 0.000,C 180.000} C_DIS
LIN {X 90.844,Y 85.304,Z 69.925,A 180.000,B 0.000,C 180.000} C_DIS
LIN {X 90.711,Y 85.376,Z 69.922,A 180.000,B 0.000,C 180.000} C_DIS
LIN {X 90.580,Y 85.451,Z 69.918,A 180.000,B 0.000,C 180.000} C_DIS
LIN {X 90.443,Y 85.530,Z 69.914,A 180.000,B 0.000,C 180.000} C_DIS
LIN {X 90.307,Y 85.608,Z 69.910,A 180.000,B 0.000,C 180.000} C_DIS
LIN {X 90.177,Y 85.682,Z 69.906,A 180.000,B 0.000,C 180.000} C_DIS
LIN {X 90.050,Y 85.759,Z 69.902,A 180.000,B 0.000,C 180.000} C_DIS
LIN {X 89.921,Y 85.843,Z 69.897,A 180.000,B 0.000,C 180.000} C_DIS
LIN {X 89.791,Y 85.927,Z 69.893,A 180.000,B 0.000,C 180.000} C_DIS
LIN {X 89.660,Y 86.013,Z 69.889,A 180.000,B 0.000,C 180.000} C_DIS
LIN {X 89.528,Y 86.098,Z 69.884,A 180.000,B 0.000,C 180.000} C_DIS
LIN {X 89.406,Y 86.181,Z 69.880,A 180.000,B 0.000,C 180.000} C_DIS
LIN {X 89.287,Y 86.268,Z 69.876,A 180.000,B 0.000,C 180.000} C_DIS
LIN {X 89.160,Y 86.360,Z 69.871,A 180.000,B 0.000,C 180.000} C_DIS
LIN {X 89.034,Y 86.453,Z 69.866,A 180.000,B 0.000,C 180.000} C_DIS
LIN {X 88.910,Y 86.543,Z 69.861,A 180.000,B 0.000,C 180.000} C_DIS
LIN {X 88.788,Y 86.635,Z 69.857,A 180.000,B 0.000,C 180.000} C_DIS
LIN {X 88.671,Y 86.731,Z 69.852,A 180.000,B 0.000,C 180.000} C_DIS
LIN {X 88.494,Y 86.876,Z 69.844,A 180.000,B 0.000,C 180.000} C_DIS
LIN {X 88.434,Y 86.925,Z 69.842,A 180.000,B 0.000,C 180.000} C_DIS
LIN {X 88.373,Y 86.975,Z 69.839,A 180.000,B 0.000,C 180.000} C_DIS
LIN {X 88.312,Y 87.025,Z 69.837,A 180.000,B 0.000,C 180.000} C_DIS
LIN {X 88.199,Y 87.119,Z 69.832,A 180.000,B 0.000,C 180.000} C_DIS
LIN {X 88.090,Y 87.218,Z 69.827,A 180.000,B 0.000,C 180.000} C_DIS
LIN {X 88.032,Y 87.271,Z 69.824,A 180.000,B 0.000,C 180.000} C_DIS
LIN {X 87.974,Y 87.325,Z 69.821,A 180.000,B 0.000,C 180.000} C_DIS
LIN {X 87.916,Y 87.378,Z 69.819,A 180.000,B 0.000,C 180.000} C_DIS
LIN {X 87.857,Y 87.431,Z 69.816,A 180.000,B 0.000,C 180.000} C_DIS
LIN {X 87.745,Y 87.533,Z 69.811,A 180.000,B 0.000,C 180.000} C_DIS
LIN {X 87.689,Y 87.585,Z 69.808,A 180.000,B 0.000,C 180.000} C_DIS
LIN {X 87.634,Y 87.637,Z 69.805,A 180.000,B 0.000,C 180.000} C_DIS
LIN {X 87.580,Y 87.691,Z 69.803,A 180.000,B 0.000,C 180.000} C_DIS
LIN {X 87.474,Y 87.800,Z 69.797,A 180.000,B 0.000,C 180.000} C_DIS
LIN {X 87.420,Y 87.855,Z 69.795,A 180.000,B 0.000,C 180.000} C_DIS
LIN {X 87.310,Y 87.967,Z 69.789,A 180.000,B 0.000,C 180.000} C_DIS
LIN {X 87.200,Y 88.080,Z 69.784,A 180.000,B 0.000,C 180.000} C_DIS
LIN {X 87.148,Y 88.133,Z 69.781,A 180.000,B 0.000,C 180.000} C_DIS
LIN {X 87.097,Y 88.187,Z 69.779,A 180.000,B 0.000,C 180.000} C_DIS
LIN {X 87.047,Y 88.242,Z 69.776,A 180.000,B 0.000,C 180.000} C_DIS
LIN {X 86.998,Y 88.297,Z 69.773,A 180.000,B 0.000,C 180.000} C_DIS
LIN {X 86.895,Y 88.415,Z 69.768,A 180.000,B 0.000,C 180.000} C_DIS
LIN {X 86.743,Y 88.590,Z 69.760,A 180.000,B 0.000,C 180.000} C_DIS
LIN {X 86.643,Y 88.704,Z 69.755,A 180.000,B 0.000,C 180.000} C_DIS
LIN {X 86.594,Y 88.761,Z 69.752,A 180.000,B 0.000,C 180.000} C_DIS
LIN {X 86.545,Y 88.821,Z 69.749,A 180.000,B 0.000,C 180.000} C_DIS
LIN {X 86.498,Y 88.882,Z 69.747,A 180.000,B 0.000,C 180.000} C_DIS
LIN {X 86.355,Y 89.065,Z 69.738,A 180.000,B 0.000,C 180.000} C_DIS
LIN {X 86.259,Y 89.189,Z 69.733,A 180.000,B 0.000,C 180.000} C_DIS
LIN {X 86.211,Y 89.250,Z 69.730,A 180.000,B 0.000,C 180.000} C_DIS
LIN {X 86.165,Y 89.310,Z 69.728,A 180.000,B 0.000,C 180.000} C_DIS
LIN {X 86.119,Y 89.369,Z 69.725,A 180.000,B 0.000,C 180.000} C_DIS
LIN {X 86.074,Y 89.429,Z 69.722,A 180.000,B 0.000,C 180.000} C_DIS
LIN {X 86.031,Y 89.490,Z 69.720,A 180.000,B 0.000,C 180.000} C_DIS
LIN {X 85.942,Y 89.619,Z 69.714,A 180.000,B 0.000,C 180.000} C_DIS
LIN {X 85.720,Y 89.939,Z 69.701,A 180.000,B 0.000,C 180.000} C_DIS
LIN {X 85.676,Y 90.003,Z 69.698,A 180.000,B 0.000,C 180.000} C_DIS
LIN {X 85.635,Y 90.066,Z 69.695,A 180.000,B 0.000,C 180.000} C_DIS
LIN {X 85.595,Y 90.130,Z 69.693,A 180.000,B 0.000,C 180.000} C_DIS
LIN {X 85.352,Y 90.527,Z 69.676,A 180.000,B 0.000,C 180.000} C_DIS
LIN {X 85.312,Y 90.592,Z 69.674,A 180.000,B 0.000,C 180.000} C_DIS
LIN {X 85.273,Y 90.656,Z 69.671,A 180.000,B 0.000,C 180.000} C_DIS
LIN {X 85.235,Y 90.721,Z 69.669,A 180.000,B 0.000,C 180.000} C_DIS
LIN {X 85.198,Y 90.787,Z 69.666,A 180.000,B 0.000,C 180.000} C_DIS
LIN {X 85.161,Y 90.856,Z 69.663,A 180.000,B 0.000,C 180.000} C_DIS
LIN {X 85.087,Y 90.992,Z 69.658,A 180.000,B 0.000,C 180.000} C_DIS
LIN {X 85.014,Y 91.129,Z 69.652,A 180.000,B 0.000,C 180.000} C_DIS
LIN {X 84.905,Y 91.333,Z 69.644,A 180.000,B 0.000,C 180.000} C_DIS
LIN {X 84.869,Y 91.400,Z 69.642,A 180.000,B 0.000,C 180.000} C_DIS
LIN {X 84.835,Y 91.468,Z 69.639,A 180.000,B 0.000,C 180.000} C_DIS
LIN {X 84.803,Y 91.537,Z 69.636,A 180.000,B 0.000,C 180.000} C_DIS
LIN {X 84.738,Y 91.678,Z 69.631,A 180.000,B 0.000,C 180.000} C_DIS
LIN {X 84.572,Y 92.032,Z 69.617,A 180.000,B 0.000,C 180.000} C_DIS
LIN {X 84.540,Y 92.102,Z 69.615,A 180.000,B 0.000,C 180.000} C_DIS
LIN {X 84.510,Y 92.174,Z 69.612,A 180.000,B 0.000,C 180.000} C_DIS
LIN {X 84.481,Y 92.244,Z 69.609,A 180.000,B 0.000,C 180.000} C_DIS
LIN {X 84.309,Y 92.674,Z 69.593,A 180.000,B 0.000,C 180.000} C_DIS
LIN {X 84.280,Y 92.746,Z 69.590,A 180.000,B 0.000,C 180.000} C_DIS
LIN {X 84.252,Y 92.817,Z 69.588,A 180.000,B 0.000,C 180.000} C_DIS
LIN {X 84.225,Y 92.888,Z 69.585,A 180.000,B 0.000,C 180.000} C_DIS
LIN {X 84.201,Y 92.959,Z 69.582,A 180.000,B 0.000,C 180.000} C_DIS
LIN {X 84.076,Y 93.329,Z 69.569,A 180.000,B 0.000,C 180.000} C_DIS
LIN {X 84.028,Y 93.472,Z 69.563,A 180.000,B 0.000,C 180.000} C_DIS
LIN {X 84.004,Y 93.544,Z 69.561,A 180.000,B 0.000,C 180.000} C_DIS
LIN {X 83.981,Y 93.617,Z 69.558,A 180.000,B 0.000,C 180.000} C_DIS
LIN {X 83.960,Y 93.692,Z 69.555,A 180.000,B 0.000,C 180.000} C_DIS
LIN {X 83.794,Y 94.294,Z 69.534,A 180.000,B 0.000,C 180.000} C_DIS
LIN {X 83.775,Y 94.367,Z 69.531,A 180.000,B 0.000,C 180.000} C_DIS
LIN {X 83.758,Y 94.440,Z 69.528,A 180.000,B 0.000,C 180.000} C_DIS
LIN {X 83.675,Y 94.821,Z 69.515,A 180.000,B 0.000,C 180.000} C_DIS
LIN {X 83.626,Y 95.051,Z 69.506,A 180.000,B 0.000,C 180.000} C_DIS
LIN {X 83.610,Y 95.128,Z 69.504,A 180.000,B 0.000,C 180.000} C_DIS
LIN {X 83.597,Y 95.203,Z 69.501,A 180.000,B 0.000,C 180.000} C_DIS
LIN {X 83.500,Y 95.813,Z 69.480,A 180.000,B 0.000,C 180.000} C_DIS
LIN {X 83.489,Y 95.888,Z 69.477,A 180.000,B 0.000,C 180.000} C_DIS
LIN {X 83.479,Y 95.963,Z 69.474,A 180.000,B 0.000,C 180.000} C_DIS
LIN {X 83.471,Y 96.039,Z 69.472,A 180.000,B 0.000,C 180.000} C_DIS
LIN {X 83.416,Y 96.586,Z 69.452,A 180.000,B 0.000,C 180.000} C_DIS
LIN {X 83.409,Y 96.664,Z 69.450,A 180.000,B 0.000,C 180.000} C_DIS
LIN {X 83.403,Y 96.740,Z 69.447,A 180.000,B 0.000,C 180.000} C_DIS
LIN {X 83.399,Y 96.816,Z 69.444,A 180.000,B 0.000,C 180.000} C_DIS
LIN {X 83.375,Y 97.360,Z 69.425,A 180.000,B 0.000,C 180.000} C_DIS
LIN {X 83.372,Y 97.437,Z 69.423,A 180.000,B 0.000,C 180.000} C_DIS
LIN {X 83.370,Y 97.514,Z 69.420,A 180.000,B 0.000,C 180.000} C_DIS
LIN {X 83.370,Y 97.591,Z 69.417,A 180.000,B 0.000,C 180.000} C_DIS
LIN {X 83.373,Y 97.824,Z 69.409,A 180.000,B 0.000,C 180.000} C_DIS
LIN {X 83.376,Y 98.059,Z 69.401,A 180.000,B 0.000,C 180.000} C_DIS
LIN {X 83.377,Y 98.215,Z 69.395,A 180.000,B 0.000,C 180.000} C_DIS
LIN {X 83.379,Y 98.292,Z 69.393,A 180.000,B 0.000,C 180.000} C_DIS
LIN {X 83.383,Y 98.368,Z 69.390,A 180.000,B 0.000,C 180.000} C_DIS
LIN {X 83.420,Y 98.913,Z 69.371,A 180.000,B 0.000,C 180.000} C_DIS
LIN {X 83.426,Y 98.990,Z 69.368,A 180.000,B 0.000,C 180.000} C_DIS
LIN {X 83.432,Y 99.067,Z 69.366,A 180.000,B 0.000,C 180.000} C_DIS
LIN {X 83.440,Y 99.143,Z 69.363,A 180.000,B 0.000,C 180.000} C_DIS
LIN {X 83.449,Y 99.221,Z 69.360,A 180.000,B 0.000,C 180.000} C_DIS
LIN {X 83.507,Y 99.686,Z 69.344,A 180.000,B 0.000,C 180.000} C_DIS
LIN {X 83.517,Y 99.764,Z 69.341,A 180.000,B 0.000,C 180.000} C_DIS
LIN {X 83.527,Y 99.840,Z 69.338,A 180.000,B 0.000,C 180.000} C_DIS
LIN {X 83.538,Y 99.916,Z 69.336,A 180.000,B 0.000,C 180.000} C_DIS
LIN {X 83.552,Y 99.992,Z 69.333,A 180.000,B 0.000,C 180.000} C_DIS
LIN {X 83.566,Y 100.068,Z 69.330,A 180.000,B 0.000,C 180.000} C_DIS
LIN {X 83.594,Y 100.223,Z 69.325,A 180.000,B 0.000,C 180.000} C_DIS
LIN {X 83.650,Y 100.529,Z 69.314,A 180.000,B 0.000,C 180.000} C_DIS
LIN {X 83.664,Y 100.605,Z 69.311,A 180.000,B 0.000,C 180.000} C_DIS
LIN {X 83.679,Y 100.681,Z 69.309,A 180.000,B 0.000,C 180.000} C_DIS
LIN {X 83.697,Y 100.757,Z 69.306,A 180.000,B 0.000,C 180.000} C_DIS
LIN {X 83.734,Y 100.909,Z 69.300,A 180.000,B 0.000,C 180.000} C_DIS
LIN {X 83.752,Y 100.986,Z 69.298,A 180.000,B 0.000,C 180.000} C_DIS
LIN {X 83.789,Y 101.139,Z 69.292,A 180.000,B 0.000,C 180.000} C_DIS
LIN {X 83.844,Y 101.367,Z 69.284,A 180.000,B 0.000,C 180.000} C_DIS
LIN {X 83.863,Y 101.441,Z 69.281,A 180.000,B 0.000,C 180.000} C_DIS
LIN {X 83.885,Y 101.515,Z 69.279,A 180.000,B 0.000,C 180.000} C_DIS
LIN {X 83.907,Y 101.589,Z 69.276,A 180.000,B 0.000,C 180.000} C_DIS
LIN {X 83.952,Y 101.740,Z 69.270,A 180.000,B 0.000,C 180.000} C_DIS
LIN {X 84.020,Y 101.966,Z 69.262,A 180.000,B 0.000,C 180.000} C_DIS
LIN {X 84.065,Y 102.116,Z 69.257,A 180.000,B 0.000,C 180.000} C_DIS
LIN {X 84.089,Y 102.191,Z 69.254,A 180.000,B 0.000,C 180.000} C_DIS
LIN {X 84.115,Y 102.264,Z 69.251,A 180.000,B 0.000,C 180.000} C_DIS
LIN {X 84.167,Y 102.409,Z 69.246,A 180.000,B 0.000,C 180.000} C_DIS
LIN {X 84.194,Y 102.482,Z 69.243,A 180.000,B 0.000,C 180.000} C_DIS
LIN {X 84.248,Y 102.630,Z 69.238,A 180.000,B 0.000,C 180.000} C_DIS
LIN {X 84.328,Y 102.851,Z 69.229,A 180.000,B 0.000,C 180.000} C_DIS
LIN {X 84.355,Y 102.924,Z 69.227,A 180.000,B 0.000,C 180.000} C_DIS
LIN {X 84.384,Y 102.996,Z 69.224,A 180.000,B 0.000,C 180.000} C_DIS
LIN {X 84.414,Y 103.067,Z 69.221,A 180.000,B 0.000,C 180.000} C_DIS
LIN {X 84.476,Y 103.211,Z 69.216,A 180.000,B 0.000,C 180.000} C_DIS
LIN {X 84.569,Y 103.428,Z 69.208,A 180.000,B 0.000,C 180.000} C_DIS
LIN {X 84.630,Y 103.572,Z 69.202,A 180.000,B 0.000,C 180.000} C_DIS
LIN {X 84.662,Y 103.644,Z 69.199,A 180.000,B 0.000,C 180.000} C_DIS
LIN {X 84.694,Y 103.715,Z 69.197,A 180.000,B 0.000,C 180.000} C_DIS
LIN {X 84.729,Y 103.784,Z 69.194,A 180.000,B 0.000,C 180.000} C_DIS
LIN {X 84.798,Y 103.924,Z 69.189,A 180.000,B 0.000,C 180.000} C_DIS
LIN {X 84.833,Y 103.994,Z 69.186,A 180.000,B 0.000,C 180.000} C_DIS
LIN {X 84.868,Y 104.065,Z 69.183,A 180.000,B 0.000,C 180.000} C_DIS
LIN {X 84.903,Y 104.135,Z 69.180,A 180.000,B 0.000,C 180.000} C_DIS
LIN {X 84.938,Y 104.206,Z 69.178,A 180.000,B 0.000,C 180.000} C_DIS
LIN {X 84.973,Y 104.276,Z 69.175,A 180.000,B 0.000,C 180.000} C_DIS
LIN {X 85.007,Y 104.345,Z 69.172,A 180.000,B 0.000,C 180.000} C_DIS
LIN {X 85.044,Y 104.414,Z 69.170,A 180.000,B 0.000,C 180.000} C_DIS
LIN {X 85.082,Y 104.482,Z 69.167,A 180.000,B 0.000,C 180.000} C_DIS
LIN {X 85.120,Y 104.550,Z 69.165,A 180.000,B 0.000,C 180.000} C_DIS
LIN {X 85.159,Y 104.619,Z 69.162,A 180.000,B 0.000,C 180.000} C_DIS
LIN {X 85.198,Y 104.687,Z 69.160,A 180.000,B 0.000,C 180.000} C_DIS
LIN {X 85.276,Y 104.823,Z 69.154,A 180.000,B 0.000,C 180.000} C_DIS
LIN {X 85.315,Y 104.892,Z 69.152,A 180.000,B 0.000,C 180.000} C_DIS
LIN {X 85.354,Y 104.960,Z 69.149,A 180.000,B 0.000,C 180.000} C_DIS
LIN {X 85.393,Y 105.028,Z 69.147,A 180.000,B 0.000,C 180.000} C_DIS
LIN {X 85.474,Y 105.161,Z 69.142,A 180.000,B 0.000,C 180.000} C_DIS
LIN {X 85.559,Y 105.292,Z 69.137,A 180.000,B 0.000,C 180.000} C_DIS
LIN {X 85.645,Y 105.424,Z 69.132,A 180.000,B 0.000,C 180.000} C_DIS
LIN {X 85.730,Y 105.556,Z 69.128,A 180.000,B 0.000,C 180.000} C_DIS
LIN {X 85.815,Y 105.687,Z 69.123,A 180.000,B 0.000,C 180.000} C_DIS
LIN {X 85.904,Y 105.816,Z 69.118,A 180.000,B 0.000,C 180.000} C_DIS
LIN {X 85.996,Y 105.943,Z 69.114,A 180.000,B 0.000,C 180.000} C_DIS
LIN {X 86.090,Y 106.070,Z 69.109,A 180.000,B 0.000,C 180.000} C_DIS
LIN {X 86.183,Y 106.197,Z 69.105,A 180.000,B 0.000,C 180.000} C_DIS
LIN {X 86.276,Y 106.324,Z 69.101,A 180.000,B 0.000,C 180.000} C_DIS
LIN {X 86.370,Y 106.448,Z 69.096,A 180.000,B 0.000,C 180.000} C_DIS
LIN {X 86.470,Y 106.569,Z 69.092,A 180.000,B 0.000,C 180.000} C_DIS
LIN {X 86.570,Y 106.691,Z 69.088,A 180.000,B 0.000,C 180.000} C_DIS
LIN {X 86.670,Y 106.812,Z 69.084,A 180.000,B 0.000,C 180.000} C_DIS
LIN {X 86.770,Y 106.933,Z 69.080,A 180.000,B 0.000,C 180.000} C_DIS
LIN {X 86.872,Y 107.053,Z 69.076,A 180.000,B 0.000,C 180.000} C_DIS
LIN {X 86.979,Y 107.168,Z 69.073,A 180.000,B 0.000,C 180.000} C_DIS
LIN {X 87.085,Y 107.283,Z 69.069,A 180.000,B 0.000,C 180.000} C_DIS
LIN {X 87.192,Y 107.399,Z 69.065,A 180.000,B 0.000,C 180.000} C_DIS
LIN {X 87.299,Y 107.514,Z 69.062,A 180.000,B 0.000,C 180.000} C_DIS
LIN {X 87.407,Y 107.628,Z 69.058,A 180.000,B 0.000,C 180.000} C_DIS
LIN {X 87.519,Y 107.737,Z 69.055,A 180.000,B 0.000,C 180.000} C_DIS
LIN {X 87.633,Y 107.847,Z 69.052,A 180.000,B 0.000,C 180.000} C_DIS
LIN {X 87.746,Y 107.956,Z 69.049,A 180.000,B 0.000,C 180.000} C_DIS
LIN {X 87.859,Y 108.065,Z 69.045,A 180.000,B 0.000,C 180.000} C_DIS
LIN {X 87.973,Y 108.173,Z 69.042,A 180.000,B 0.000,C 180.000} C_DIS
LIN {X 88.092,Y 108.276,Z 69.040,A 180.000,B 0.000,C 180.000} C_DIS
LIN {X 88.212,Y 108.379,Z 69.037,A 180.000,B 0.000,C 180.000} C_DIS
LIN {X 88.331,Y 108.481,Z 69.034,A 180.000,B 0.000,C 180.000} C_DIS
LIN {X 88.451,Y 108.584,Z 69.031,A 180.000,B 0.000,C 180.000} C_DIS
LIN {X 88.694,Y 108.782,Z 69.026,A 180.000,B 0.000,C 180.000} C_DIS
LIN {X 88.945,Y 108.973,Z 69.022,A 180.000,B 0.000,C 180.000} C_DIS
LIN {X 89.196,Y 109.164,Z 69.018,A 180.000,B 0.000,C 180.000} C_DIS
LIN {X 89.455,Y 109.341,Z 69.014,A 180.000,B 0.000,C 180.000} C_DIS
LIN {X 89.716,Y 109.517,Z 69.011,A 180.000,B 0.000,C 180.000} C_DIS
LIN {X 89.981,Y 109.688,Z 69.008,A 180.000,B 0.000,C 180.000} C_DIS
LIN {X 90.252,Y 109.849,Z 69.005,A 180.000,B 0.000,C 180.000} C_DIS
LIN {X 90.522,Y 110.010,Z 69.003,A 180.000,B 0.000,C 180.000} C_DIS
LIN {X 90.800,Y 110.158,Z 69.002,A 180.000,B 0.000,C 180.000} C_DIS
LIN {X 91.080,Y 110.303,Z 69.001,A 180.000,B 0.000,C 180.000} C_DIS
LIN {X 91.362,Y 110.443,Z 69.000,A 180.000,B 0.000,C 180.000} C_DIS
LIN {X 91.561,Y 110.532,Z 69.000,A 180.000,B 0.000,C 180.000} C_DIS
; Cutting Move Starts
LIN {X 91.891,Y 110.680,Z 69.000,A 180.000,B 0.000,C 180.000} C_DIS
LIN {X 92.070,Y 110.757,Z 69.000,A 180.000,B 0.000,C 180.000} C_DIS
LIN {X 92.249,Y 110.825,Z 69.000,A 180.000,B 0.000,C 180.000} C_DIS
LIN {X 92.606,Y 110.961,Z 69.000,A 180.000,B 0.000,C 180.000} C_DIS
LIN {X 92.761,Y 111.019,Z 69.000,A 180.000,B 0.000,C 180.000} C_DIS
LIN {X 92.785,Y 111.028,Z 69.000,A 180.000,B 0.000,C 180.000} C_DIS
LIN {X 92.964,Y 111.085,Z 69.000,A 180.000,B 0.000,C 180.000} C_DIS
LIN {X 93.321,Y 111.199,Z 69.000,A 180.000,B 0.000,C 180.000} C_DIS
LIN {X 93.500,Y 111.256,Z 69.000,A 180.000,B 0.000,C 180.000} C_DIS
LIN {X 93.679,Y 111.305,Z 69.000,A 180.000,B 0.000,C 180.000} C_DIS
LIN {X 94.215,Y 111.443,Z 69.000,A 180.000,B 0.000,C 180.000} C_DIS
LIN {X 94.394,Y 111.484,Z 69.000,A 180.000,B 0.000,C 180.000} C_DIS
LIN {X 94.930,Y 111.591,Z 69.000,A 180.000,B 0.000,C 180.000} C_DIS
LIN {X 95.109,Y 111.625,Z 69.000,A 180.000,B 0.000,C 180.000} C_DIS
LIN {X 95.288,Y 111.651,Z 69.000,A 180.000,B 0.000,C 180.000} C_DIS
LIN {X 95.824,Y 111.727,Z 69.000,A 180.000,B 0.000,C 180.000} C_DIS
LIN {X 95.882,Y 111.734,Z 69.000,A 180.000,B 0.000,C 180.000} C_DIS
LIN {X 96.003,Y 111.746,Z 69.000,A 180.000,B 0.000,C 180.000} C_DIS
LIN {X 96.539,Y 111.791,Z 69.000,A 180.000,B 0.000,C 180.000} C_DIS
LIN {X 96.718,Y 111.805,Z 69.000,A 180.000,B 0.000,C 180.000} C_DIS
LIN {X 96.897,Y 111.810,Z 69.000,A 180.000,B 0.000,C 180.000} C_DIS
LIN {X 97.433,Y 111.825,Z 69.000,A 180.000,B 0.000,C 180.000} C_DIS
LIN {X 97.612,Y 111.824,Z 69.000,A 180.000,B 0.000,C 180.000} C_DIS
LIN {X 98.148,Y 111.809,Z 69.000,A 180.000,B 0.000,C 180.000} C_DIS
LIN {X 98.327,Y 111.802,Z 69.000,A 180.000,B 0.000,C 180.000} C_DIS
LIN {X 98.505,Y 111.787,Z 69.000,A 180.000,B 0.000,C 180.000} C_DIS
LIN {X 99.042,Y 111.742,Z 69.000,A 180.000,B 0.000,C 180.000} C_DIS
LIN {X 99.118,Y 111.734,Z 69.000,A 180.000,B 0.000,C 180.000} C_DIS
LIN {X 99.221,Y 111.721,Z 69.000,A 180.000,B 0.000,C 180.000} C_DIS
LIN {X 99.757,Y 111.645,Z 69.000,A 180.000,B 0.000,C 180.000} C_DIS
LIN {X 99.936,Y 111.617,Z 69.000,A 180.000,B 0.000,C 180.000} C_DIS
LIN {X 100.114,Y 111.582,Z 69.000,A 180.000,B 0.000,C 180.000} C_DIS
LIN {X 100.472,Y 111.511,Z 69.000,A 180.000,B 0.000,C 180.000} C_DIS
LIN {X 100.651,Y 111.475,Z 69.000,A 180.000,B 0.000,C 180.000} C_DIS
LIN {X 100.829,Y 111.432,Z 69.000,A 180.000,B 0.000,C 180.000} C_DIS
LIN {X 101.366,Y 111.293,Z 69.000,A 180.000,B 0.000,C 180.000} C_DIS
LIN {X 101.545,Y 111.242,Z 69.000,A 180.000,B 0.000,C 180.000} C_DIS
LIN {X 102.081,Y 111.071,Z 69.000,A 180.000,B 0.000,C 180.000} C_DIS
LIN {X 102.239,Y 111.019,Z 69.000,A 180.000,B 0.000,C 180.000} C_DIS
LIN {X 102.260,Y 111.012,Z 69.000,A 180.000,B 0.000,C 180.000} C_DIS
LIN {X 102.438,Y 110.944,Z 69.000,A 180.000,B 0.000,C 180.000} C_DIS
LIN {X 102.796,Y 110.808,Z 69.000,A 180.000,B 0.000,C 180.000} C_DIS
LIN {X 102.975,Y 110.739,Z 69.000,A 180.000,B 0.000,C 180.000} C_DIS
LIN {X 103.150,Y 110.662,Z 69.000,A 180.000,B 0.000,C 180.000} C_DIS
LIN {X 103.549,Y 110.483,Z 69.000,A 180.000,B 0.000,C 180.000} C_DIS
LIN {X 103.690,Y 110.419,Z 69.000,A 180.000,B 0.000,C 180.000} C_DIS
LIN {X 103.869,Y 110.330,Z 69.000,A 180.000,B 0.000,C 180.000} C_DIS
LIN {X 104.264,Y 110.126,Z 69.000,A 180.000,B 0.000,C 180.000} C_DIS
LIN {X 104.405,Y 110.052,Z 69.000,A 180.000,B 0.000,C 180.000} C_DIS
LIN {X 104.584,Y 109.949,Z 69.000,A 180.000,B 0.000,C 180.000} C_DIS
LIN {X 104.941,Y 109.738,Z 69.000,A 180.000,B 0.000,C 180.000} C_DIS
LIN {X 105.120,Y 109.631,Z 69.000,A 180.000,B 0.000,C 180.000} C_DIS
LIN {X 105.185,Y 109.589,Z 69.000,A 180.000,B 0.000,C 180.000} C_DIS
LIN {X 105.477,Y 109.394,Z 69.000,A 180.000,B 0.000,C 180.000} C_DIS
LIN {X 105.720,Y 109.232,Z 69.000,A 180.000,B 0.000,C 180.000} C_DIS
LIN {X 105.835,Y 109.151,Z 69.000,A 180.000,B 0.000,C 180.000} C_DIS
LIN {X 105.966,Y 109.053,Z 69.000,A 180.000,B 0.000,C 180.000} C_DIS
LIN {X 106.371,Y 108.748,Z 69.000,A 180.000,B 0.000,C 180.000} C_DIS
LIN {X 106.438,Y 108.695,Z 69.000,A 180.000,B 0.000,C 180.000} C_DIS
LIN {X 106.550,Y 108.602,Z 69.000,A 180.000,B 0.000,C 180.000} C_DIS
LIN {X 106.908,Y 108.300,Z 69.000,A 180.000,B 0.000,C 180.000} C_DIS
LIN {X 107.072,Y 108.159,Z 69.000,A 180.000,B 0.000,C 180.000} C_DIS
LIN {X 107.086,Y 108.145,Z 69.000,A 180.000,B 0.000,C 180.000} C_DIS
LIN {X 107.265,Y 107.977,Z 69.000,A 180.000,B 0.000,C 180.000} C_DIS
LIN {X 107.450,Y 107.802,Z 69.000,A 180.000,B 0.000,C 180.000} C_DIS
LIN {X 107.623,Y 107.637,Z 69.000,A 180.000,B 0.000,C 180.000} C_DIS
LIN {X 107.637,Y 107.623,Z 69.000,A 180.000,B 0.000,C 180.000} C_DIS
LIN {X 107.802,Y 107.450,Z 69.000,A 180.000,B 0.000,C 180.000} C_DIS
LIN {X 107.980,Y 107.261,Z 69.000,A 180.000,B 0.000,C 180.000} C_DIS
LIN {X 108.145,Y 107.086,Z 69.000,A 180.000,B 0.000,C 180.000} C_DIS
LIN {X 108.159,Y 107.071,Z 69.000,A 180.000,B 0.000,C 180.000} C_DIS
LIN {X 108.301,Y 106.908,Z 69.000,A 180.000,B 0.000,C 180.000} C_DIS
LIN {X 108.602,Y 106.550,Z 69.000,A 180.000,B 0.000,C 180.000} C_DIS
LIN {X 108.695,Y 106.439,Z 69.000,A 180.000,B 0.000,C 180.000} C_DIS
LIN {X 108.748,Y 106.371,Z 69.000,A 180.000,B 0.000,C 180.000} C_DIS
LIN {X 109.053,Y 105.966,Z 69.000,A 180.000,B 0.000,C 180.000} C_DIS
LIN {X 109.151,Y 105.835,Z 69.000,A 180.000,B 0.000,C 180.000} C_DIS
LIN {X 109.232,Y 105.720,Z 69.000,A 180.000,B 0.000,C 180.000} C_DIS
LIN {X 109.589,Y 105.185,Z 69.000,A 180.000,B 0.000,C 180.000} C_DIS
LIN {X 109.632,Y 105.120,Z 69.000,A 180.000,B 0.000,C 180.000} C_DIS
LIN {X 109.738,Y 104.941,Z 69.000,A 180.000,B 0.000,C 180.000} C_DIS
LIN {X 109.949,Y 104.584,Z 69.000,A 180.000,B 0.000,C 180.000} C_DIS
LIN {X 110.052,Y 104.405,Z 69.000,A 180.000,B 0.000,C 180.000} C_DIS
LIN {X 110.126,Y 104.264,Z 69.000,A 180.000,B 0.000,C 180.000} C_DIS
LIN {X 110.330,Y 103.869,Z 69.000,A 180.000,B 0.000,C 180.000} C_DIS
LIN {X 110.420,Y 103.690,Z 69.000,A 180.000,B 0.000,C 180.000} C_DIS
LIN {X 110.483,Y 103.549,Z 69.000,A 180.000,B 0.000,C 180.000} C_DIS
LIN {X 110.662,Y 103.150,Z 69.000,A 180.000,B 0.000,C 180.000} C_DIS
LIN {X 110.739,Y 102.975,Z 69.000,A 180.000,B 0.000,C 180.000} C_DIS
LIN {X 110.808,Y 102.796,Z 69.000,A 180.000,B 0.000,C 180.000} C_DIS
LIN {X 110.944,Y 102.438,Z 69.000,A 180.000,B 0.000,C 180.000} C_DIS
LIN {X 111.012,Y 102.260,Z 69.000,A 180.000,B 0.000,C 180.000} C_DIS
LIN {X 111.019,Y 102.240,Z 69.000,A 180.000,B 0.000,C 180.000} C_DIS
LIN {X 111.071,Y 102.081,Z 69.000,A 180.000,B 0.000,C 180.000} C_DIS
LIN {X 111.242,Y 101.545,Z 69.000,A 180.000,B 0.000,C 180.000} C_DIS
LIN {X 111.293,Y 101.366,Z 69.000,A 180.000,B 0.000,C 180.000} C_DIS
LIN {X 111.431,Y 100.829,Z 69.000,A 180.000,B 0.000,C 180.000} C_DIS
LIN {X 111.475,Y 100.651,Z 69.000,A 180.000,B 0.000,C 180.000} C_DIS
LIN {X 111.511,Y 100.472,Z 69.000,A 180.000,B 0.000,C 180.000} C_DIS
LIN {X 111.582,Y 100.114,Z 69.000,A 180.000,B 0.000,C 180.000} C_DIS
LIN {X 111.617,Y 99.936,Z 69.000,A 180.000,B 0.000,C 180.000} C_DIS
LIN {X 111.645,Y 99.757,Z 69.000,A 180.000,B 0.000,C 180.000} C_DIS
LIN {X 111.720,Y 99.221,Z 69.000,A 180.000,B 0.000,C 180.000} C_DIS
LIN {X 111.734,Y 99.116,Z 69.000,A 180.000,B 0.000,C 180.000} C_DIS
LIN {X 111.742,Y 99.042,Z 69.000,A 180.000,B 0.000,C 180.000} C_DIS
LIN {X 111.757,Y 98.863,Z 69.000,A 180.000,B 0.000,C 180.000} C_DIS
LIN {X 111.788,Y 98.505,Z 69.000,A 180.000,B 0.000,C 180.000} C_DIS
LIN {X 111.802,Y 98.327,Z 69.000,A 180.000,B 0.000,C 180.000} C_DIS
LIN {X 111.809,Y 98.148,Z 69.000,A 180.000,B 0.000,C 180.000} C_DIS
LIN {X 111.824,Y 97.612,Z 69.000,A 180.000,B 0.000,C 180.000} C_DIS
LIN {X 111.825,Y 97.433,Z 69.000,A 180.000,B 0.000,C 180.000} C_DIS
LIN {X 111.820,Y 97.254,Z 69.000,A 180.000,B 0.000,C 180.000} C_DIS
LIN {X 111.810,Y 96.897,Z 69.000,A 180.000,B 0.000,C 180.000} C_DIS
LIN {X 111.805,Y 96.718,Z 69.000,A 180.000,B 0.000,C 180.000} C_DIS
LIN {X 111.791,Y 96.539,Z 69.000,A 180.000,B 0.000,C 180.000} C_DIS
LIN {X 111.746,Y 96.003,Z 69.000,A 180.000,B 0.000,C 180.000} C_DIS
LIN {X 111.734,Y 95.884,Z 69.000,A 180.000,B 0.000,C 180.000} C_DIS
LIN {X 111.727,Y 95.824,Z 69.000,A 180.000,B 0.000,C 180.000} C_DIS
LIN {X 111.702,Y 95.645,Z 69.000,A 180.000,B 0.000,C 180.000} C_DIS
LIN {X 111.651,Y 95.288,Z 69.000,A 180.000,B 0.000,C 180.000} C_DIS
LIN {X 111.625,Y 95.109,Z 69.000,A 180.000,B 0.000,C 180.000} C_DIS
LIN {X 111.591,Y 94.930,Z 69.000,A 180.000,B 0.000,C 180.000} C_DIS
LIN {X 111.484,Y 94.394,Z 69.000,A 180.000,B 0.000,C 180.000} C_DIS
LIN {X 111.443,Y 94.215,Z 69.000,A 180.000,B 0.000,C 180.000} C_DIS
LIN {X 111.304,Y 93.679,Z 69.000,A 180.000,B 0.000,C 180.000} C_DIS
LIN {X 111.256,Y 93.500,Z 69.000,A 180.000,B 0.000,C 180.000} C_DIS
LIN {X 111.200,Y 93.321,Z 69.000,A 180.000,B 0.000,C 180.000} C_DIS
LIN {X 111.086,Y 92.964,Z 69.000,A 180.000,B 0.000,C 180.000} C_DIS
LIN {X 111.028,Y 92.785,Z 69.000,A 180.000,B 0.000,C 180.000} C_DIS
LIN {X 111.019,Y 92.760,Z 69.000,A 180.000,B 0.000,C 180.000} C_DIS
LIN {X 110.961,Y 92.606,Z 69.000,A 180.000,B 0.000,C 180.000} C_DIS
LIN {X 110.825,Y 92.249,Z 69.000,A 180.000,B 0.000,C 180.000} C_DIS
LIN {X 110.756,Y 92.070,Z 69.000,A 180.000,B 0.000,C 180.000} C_DIS
LIN {X 110.680,Y 91.891,Z 69.000,A 180.000,B 0.000,C 180.000} C_DIS
LIN {X 110.440,Y 91.355,Z 69.000,A 180.000,B 0.000,C 180.000} C_DIS
LIN {X 110.353,Y 91.176,Z 69.000,A 180.000,B 0.000,C 180.000} C_DIS
LIN {X 110.076,Y 90.640,Z 69.000,A 180.000,B 0.000,C 180.000} C_DIS
LIN {X 109.975,Y 90.461,Z 69.000,A 180.000,B 0.000,C 180.000} C_DIS
LIN {X 109.764,Y 90.103,Z 69.000,A 180.000,B 0.000,C 180.000} C_DIS
LIN {X 109.659,Y 89.925,Z 69.000,A 180.000,B 0.000,C 180.000} C_DIS
LIN {X 109.589,Y 89.815,Z 69.000,A 180.000,B 0.000,C 180.000} C_DIS
LIN {X 109.232,Y 89.280,Z 69.000,A 180.000,B 0.000,C 180.000} C_DIS
LIN {X 109.183,Y 89.209,Z 69.000,A 180.000,B 0.000,C 180.000} C_DIS
LIN {X 109.053,Y 89.034,Z 69.000,A 180.000,B 0.000,C 180.000} C_DIS
LIN {X 108.781,Y 88.673,Z 69.000,A 180.000,B 0.000,C 180.000} C_DIS
LIN {X 108.695,Y 88.561,Z 69.000,A 180.000,B 0.000,C 180.000} C_DIS
LIN {X 108.640,Y 88.494,Z 69.000,A 180.000,B 0.000,C 180.000} C_DIS
LIN {X 108.338,Y 88.137,Z 69.000,A 180.000,B 0.000,C 180.000} C_DIS
LIN {X 108.186,Y 87.958,Z 69.000,A 180.000,B 0.000,C 180.000} C_DIS
LIN {X 108.159,Y 87.929,Z 69.000,A 180.000,B 0.000,C 180.000} C_DIS
LIN {X 108.018,Y 87.779,Z 69.000,A 180.000,B 0.000,C 180.000} C_DIS
LIN {X 107.680,Y 87.422,Z 69.000,A 180.000,B 0.000,C 180.000} C_DIS
LIN {X 107.623,Y 87.363,Z 69.000,A 180.000,B 0.000,C 180.000} C_DIS
LIN {X 107.497,Y 87.243,Z 69.000,A 180.000,B 0.000,C 180.000} C_DIS
LIN {X 107.119,Y 86.885,Z 69.000,A 180.000,B 0.000,C 180.000} C_DIS
LIN {X 107.086,Y 86.855,Z 69.000,A 180.000,B 0.000,C 180.000} C_DIS
LIN {X 106.916,Y 86.707,Z 69.000,A 180.000,B 0.000,C 180.000} C_DIS
LIN {X 106.550,Y 86.398,Z 69.000,A 180.000,B 0.000,C 180.000} C_DIS
LIN {X 106.492,Y 86.349,Z 69.000,A 180.000,B 0.000,C 180.000} C_DIS
LIN {X 106.371,Y 86.252,Z 69.000,A 180.000,B 0.000,C 180.000} C_DIS
LIN {X 106.014,Y 85.983,Z 69.000,A 180.000,B 0.000,C 180.000} C_DIS
LIN {X 105.835,Y 85.849,Z 69.000,A 180.000,B 0.000,C 180.000} C_DIS
LIN {X 105.785,Y 85.813,Z 69.000,A 180.000,B 0.000,C 180.000} C_DIS
LIN {X 105.656,Y 85.726,Z 69.000,A 180.000,B 0.000,C 180.000} C_DIS
LIN {X 105.252,Y 85.455,Z 69.000,A 180.000,B 0.000,C 180.000} C_DIS
LIN {X 105.120,Y 85.369,Z 69.000,A 180.000,B 0.000,C 180.000} C_DIS
LIN {X 104.966,Y 85.276,Z 69.000,A 180.000,B 0.000,C 180.000} C_DIS
LIN {X 104.584,Y 85.051,Z 69.000,A 180.000,B 0.000,C 180.000} C_DIS
LIN {X 104.405,Y 84.948,Z 69.000,A 180.000,B 0.000,C 180.000} C_DIS
LIN {X 104.350,Y 84.919,Z 69.000,A 180.000,B 0.000,C 180.000} C_DIS
LIN {X 103.869,Y 84.670,Z 69.000,A 180.000,B 0.000,C 180.000} C_DIS
LIN {X 103.690,Y 84.581,Z 69.000,A 180.000,B 0.000,C 180.000} C_DIS
LIN {X 103.648,Y 84.561,Z 69.000,A 180.000,B 0.000,C 180.000} C_DIS
LIN {X 103.511,Y 84.500,Z 69.000,A 180.000,B 0.000,C 180.000} C_DIS
LIN {X 103.153,Y 84.340,Z 69.000,A 180.000,B 0.000,C 180.000} C_DIS
LIN {X 102.975,Y 84.261,Z 69.000,A 180.000,B 0.000,C 180.000} C_DIS
LIN {X 102.827,Y 84.204,Z 69.000,A 180.000,B 0.000,C 180.000} C_DIS
LIN {X 102.358,Y 84.025,Z 69.000,A 180.000,B 0.000,C 180.000} C_DIS
LIN {X 102.260,Y 83.988,Z 69.000,A 180.000,B 0.000,C 180.000} C_DIS
LIN {X 102.081,Y 83.929,Z 69.000,A 180.000,B 0.000,C 180.000} C_DIS
LIN {X 101.545,Y 83.758,Z 69.000,A 180.000,B 0.000,C 180.000} C_DIS
LIN {X 101.366,Y 83.707,Z 69.000,A 180.000,B 0.000,C 180.000} C_DIS
LIN {X 100.829,Y 83.568,Z 69.000,A 180.000,B 0.000,C 180.000} C_DIS
LIN {X 100.651,Y 83.525,Z 69.000,A 180.000,B 0.000,C 180.000} C_DIS
LIN {X 100.470,Y 83.489,Z 69.000,A 180.000,B 0.000,C 180.000} C_DIS
LIN {X 100.114,Y 83.418,Z 69.000,A 180.000,B 0.000,C 180.000} C_DIS
LIN {X 99.936,Y 83.383,Z 69.000,A 180.000,B 0.000,C 180.000} C_DIS
LIN {X 99.757,Y 83.355,Z 69.000,A 180.000,B 0.000,C 180.000} C_DIS
LIN {X 99.221,Y 83.279,Z 69.000,A 180.000,B 0.000,C 180.000} C_DIS
LIN {X 99.042,Y 83.258,Z 69.000,A 180.000,B 0.000,C 180.000} C_DIS
LIN {X 98.505,Y 83.213,Z 69.000,A 180.000,B 0.000,C 180.000} C_DIS
LIN {X 98.327,Y 83.198,Z 69.000,A 180.000,B 0.000,C 180.000} C_DIS
LIN {X 98.148,Y 83.191,Z 69.000,A 180.000,B 0.000,C 180.000} C_DIS
LIN {X 97.612,Y 83.176,Z 69.000,A 180.000,B 0.000,C 180.000} C_DIS
LIN {X 97.433,Y 83.175,Z 69.000,A 180.000,B 0.000,C 180.000} C_DIS
LIN {X 96.897,Y 83.190,Z 69.000,A 180.000,B 0.000,C 180.000} C_DIS
LIN {X 96.718,Y 83.195,Z 69.000,A 180.000,B 0.000,C 180.000} C_DIS
LIN {X 96.539,Y 83.209,Z 69.000,A 180.000,B 0.000,C 180.000} C_DIS
LIN {X 96.003,Y 83.254,Z 69.000,A 180.000,B 0.000,C 180.000} C_DIS
LIN {X 95.824,Y 83.273,Z 69.000,A 180.000,B 0.000,C 180.000} C_DIS
LIN {X 95.288,Y 83.349,Z 69.000,A 180.000,B 0.000,C 180.000} C_DIS
LIN {X 95.109,Y 83.375,Z 69.000,A 180.000,B 0.000,C 180.000} C_DIS
LIN {X 94.930,Y 83.409,Z 69.000,A 180.000,B 0.000,C 180.000} C_DIS
LIN {X 94.394,Y 83.516,Z 69.000,A 180.000,B 0.000,C 180.000} C_DIS
LIN {X 94.215,Y 83.557,Z 69.000,A 180.000,B 0.000,C 180.000} C_DIS
LIN {X 93.679,Y 83.695,Z 69.000,A 180.000,B 0.000,C 180.000} C_DIS
LIN {X 93.500,Y 83.744,Z 69.000,A 180.000,B 0.000,C 180.000} C_DIS
LIN {X 93.321,Y 83.801,Z 69.000,A 180.000,B 0.000,C 180.000} C_DIS
LIN {X 92.964,Y 83.915,Z 69.000,A 180.000,B 0.000,C 180.000} C_DIS
LIN {X 92.785,Y 83.972,Z 69.000,A 180.000,B 0.000,C 180.000} C_DIS
LIN {X 92.642,Y 84.025,Z 69.000,A 180.000,B 0.000,C 180.000} C_DIS
LIN {X 92.173,Y 84.204,Z 69.000,A 180.000,B 0.000,C 180.000} C_DIS
LIN {X 92.070,Y 84.243,Z 69.000,A 180.000,B 0.000,C 180.000} C_DIS
LIN {X 91.891,Y 84.320,Z 69.000,A 180.000,B 0.000,C 180.000} C_DIS
LIN {X 91.355,Y 84.560,Z 69.000,A 180.000,B 0.000,C 180.000} C_DIS
LIN {X 91.352,Y 84.561,Z 69.000,A 180.000,B 0.000,C 180.000} C_DIS
LIN {X 91.176,Y 84.647,Z 69.000,A 180.000,B 0.000,C 180.000} C_DIS
LIN {X 90.640,Y 84.924,Z 69.000,A 180.000,B 0.000,C 180.000} C_DIS
LIN {X 90.461,Y 85.025,Z 69.000,A 180.000,B 0.000,C 180.000} C_DIS
LIN {X 90.034,Y 85.276,Z 69.000,A 180.000,B 0.000,C 180.000} C_DIS
LIN {X 89.925,Y 85.341,Z 69.000,A 180.000,B 0.000,C 180.000} C_DIS
LIN {X 89.748,Y 85.455,Z 69.000,A 180.000,B 0.000,C 180.000} C_DIS
LIN {X 89.388,Y 85.696,Z 69.000,A 180.000,B 0.000,C 180.000} C_DIS
LIN {X 89.215,Y 85.813,Z 69.000,A 180.000,B 0.000,C 180.000} C_DIS
LIN {X 89.209,Y 85.816,Z 69.000,A 180.000,B 0.000,C 180.000} C_DIS
LIN {X 89.031,Y 85.950,Z 69.000,A 180.000,B 0.000,C 180.000} C_DIS
LIN {X 88.673,Y 86.219,Z 69.000,A 180.000,B 0.000,C 180.000} C_DIS
LIN {X 88.508,Y 86.349,Z 69.000,A 180.000,B 0.000,C 180.000} C_DIS
LIN {X 88.494,Y 86.360,Z 69.000,A 180.000,B 0.000,C 180.000} C_DIS
LIN {X 88.084,Y 86.707,Z 69.000,A 180.000,B 0.000,C 180.000} C_DIS
LIN {X 87.958,Y 86.814,Z 69.000,A 180.000,B 0.000,C 180.000} C_DIS
LIN {X 87.881,Y 86.885,Z 69.000,A 180.000,B 0.000,C 180.000} C_DIS
LIN {X 87.422,Y 87.319,Z 69.000,A 180.000,B 0.000,C 180.000} C_DIS
LIN {X 87.320,Y 87.422,Z 69.000,A 180.000,B 0.000,C 180.000} C_DIS
LIN {X 86.885,Y 87.881,Z 69.000,A 180.000,B 0.000,C 180.000} C_DIS
LIN {X 86.814,Y 87.958,Z 69.000,A 180.000,B 0.000,C 180.000} C_DIS
LIN {X 86.707,Y 88.084,Z 69.000,A 180.000,B 0.000,C 180.000} C_DIS
LIN {X 86.349,Y 88.507,Z 69.000,A 180.000,B 0.000,C 180.000} C_DIS
LIN {X 86.219,Y 88.673,Z 69.000,A 180.000,B 0.000,C 180.000} C_DIS
LIN {X 85.950,Y 89.031,Z 69.000,A 180.000,B 0.000,C 180.000} C_DIS
LIN {X 85.817,Y 89.209,Z 69.000,A 180.000,B 0.000,C 180.000} C_DIS
LIN {X 85.813,Y 89.215,Z 69.000,A 180.000,B 0.000,C 180.000} C_DIS
LIN {X 85.696,Y 89.388,Z 69.000,A 180.000,B 0.000,C 180.000} C_DIS
LIN {X 85.455,Y 89.748,Z 69.000,A 180.000,B 0.000,C 180.000} C_DIS
LIN {X 85.341,Y 89.925,Z 69.000,A 180.000,B 0.000,C 180.000} C_DIS
LIN {X 85.276,Y 90.034,Z 69.000,A 180.000,B 0.000,C 180.000} C_DIS
LIN {X 85.025,Y 90.461,Z 69.000,A 180.000,B 0.000,C 180.000} C_DIS
LIN {X 84.924,Y 90.640,Z 69.000,A 180.000,B 0.000,C 180.000} C_DIS
LIN {X 84.647,Y 91.176,Z 69.000,A 180.000,B 0.000,C 180.000} C_DIS
LIN {X 84.561,Y 91.351,Z 69.000,A 180.000,B 0.000,C 180.000} C_DIS
LIN {X 84.320,Y 91.891,Z 69.000,A 180.000,B 0.000,C 180.000} C_DIS
LIN {X 84.244,Y 92.070,Z 69.000,A 180.000,B 0.000,C 180.000} C_DIS
LIN {X 84.204,Y 92.174,Z 69.000,A 180.000,B 0.000,C 180.000} C_DIS
LIN {X 84.025,Y 92.642,Z 69.000,A 180.000,B 0.000,C 180.000} C_DIS
LIN {X 83.972,Y 92.785,Z 69.000,A 180.000,B 0.000,C 180.000} C_DIS
LIN {X 83.914,Y 92.964,Z 69.000,A 180.000,B 0.000,C 180.000} C_DIS
LIN {X 83.800,Y 93.321,Z 69.000,A 180.000,B 0.000,C 180.000} C_DIS
LIN {X 83.744,Y 93.500,Z 69.000,A 180.000,B 0.000,C 180.000} C_DIS
LIN {X 83.696,Y 93.679,Z 69.000,A 180.000,B 0.000,C 180.000} C_DIS
LIN {X 83.557,Y 94.215,Z 69.000,A 180.000,B 0.000,C 180.000} C_DIS
LIN {X 83.516,Y 94.394,Z 69.000,A 180.000,B 0.000,C 180.000} C_DIS
LIN {X 83.409,Y 94.930,Z 69.000,A 180.000,B 0.000,C 180.000} C_DIS
LIN {X 83.375,Y 95.109,Z 69.000,A 180.000,B 0.000,C 180.000} C_DIS
LIN {X 83.349,Y 95.288,Z 69.000,A 180.000,B 0.000,C 180.000} C_DIS
LIN {X 83.310,Y 95.563,Z 69.000,A 180.000,B 0.000,C 180.000} C_DIS
LIN {X 83.298,Y 95.645,Z 69.000,A 180.000,B 0.000,C 180.000} C_DIS
LIN {X 83.276,Y 95.804,Z 69.000,A 180.000,B 0.000,C 180.000} C_DIS
LIN {X 83.273,Y 95.824,Z 69.000,A 180.000,B 0.000,C 180.000} C_DIS
LIN {X 83.254,Y 96.003,Z 69.000,A 180.000,B 0.000,C 180.000} C_DIS
LIN {X 83.209,Y 96.539,Z 69.000,A 180.000,B 0.000,C 180.000} C_DIS
LIN {X 83.195,Y 96.718,Z 69.000,A 180.000,B 0.000,C 180.000} C_DIS
LIN {X 83.190,Y 96.897,Z 69.000,A 180.000,B 0.000,C 180.000} C_DIS
LIN {X 83.180,Y 97.254,Z 69.000,A 180.000,B 0.000,C 180.000} C_DIS
LIN {X 83.175,Y 97.433,Z 69.000,A 180.000,B 0.000,C 180.000} C_DIS
LIN {X 83.176,Y 97.612,Z 69.000,A 180.000,B 0.000,C 180.000} C_DIS
LIN {X 83.191,Y 98.148,Z 69.000,A 180.000,B 0.000,C 180.000} C_DIS
LIN {X 83.198,Y 98.327,Z 69.000,A 180.000,B 0.000,C 180.000} C_DIS
LIN {X 83.212,Y 98.505,Z 69.000,A 180.000,B 0.000,C 180.000} C_DIS
LIN {X 83.243,Y 98.863,Z 69.000,A 180.000,B 0.000,C 180.000} C_DIS
LIN {X 83.258,Y 99.042,Z 69.000,A 180.000,B 0.000,C 180.000} C_DIS
LIN {X 83.280,Y 99.221,Z 69.000,A 180.000,B 0.000,C 180.000} C_DIS
LIN {X 83.355,Y 99.757,Z 69.000,A 180.000,B 0.000,C 180.000} C_DIS
LIN {X 83.383,Y 99.936,Z 69.000,A 180.000,B 0.000,C 180.000} C_DIS
LIN {X 83.418,Y 100.114,Z 69.000,A 180.000,B 0.000,C 180.000} C_DIS
LIN {X 83.489,Y 100.472,Z 69.000,A 180.000,B 0.000,C 180.000} C_DIS
LIN {X 83.525,Y 100.651,Z 69.000,A 180.000,B 0.000,C 180.000} C_DIS
LIN {X 83.569,Y 100.829,Z 69.000,A 180.000,B 0.000,C 180.000} C_DIS
LIN {X 83.707,Y 101.366,Z 69.000,A 180.000,B 0.000,C 180.000} C_DIS
LIN {X 83.758,Y 101.545,Z 69.000,A 180.000,B 0.000,C 180.000} C_DIS
LIN {X 83.929,Y 102.081,Z 69.000,A 180.000,B 0.000,C 180.000} C_DIS
LIN {X 83.988,Y 102.260,Z 69.000,A 180.000,B 0.000,C 180.000} C_DIS
LIN {X 84.025,Y 102.358,Z 69.000,A 180.000,B 0.000,C 180.000} C_DIS
LIN {X 84.204,Y 102.826,Z 69.000,A 180.000,B 0.000,C 180.000} C_DIS
LIN {X 84.261,Y 102.975,Z 69.000,A 180.000,B 0.000,C 180.000} C_DIS
LIN {X 84.340,Y 103.153,Z 69.000,A 180.000,B 0.000,C 180.000} C_DIS
LIN {X 84.561,Y 103.649,Z 69.000,A 180.000,B 0.000,C 180.000} C_DIS
LIN {X 84.580,Y 103.690,Z 69.000,A 180.000,B 0.000,C 180.000} C_DIS
LIN {X 84.670,Y 103.869,Z 69.000,A 180.000,B 0.000,C 180.000} C_DIS
LIN {X 84.919,Y 104.350,Z 69.000,A 180.000,B 0.000,C 180.000} C_DIS
LIN {X 84.948,Y 104.405,Z 69.000,A 180.000,B 0.000,C 180.000} C_DIS
LIN {X 85.051,Y 104.584,Z 69.000,A 180.000,B 0.000,C 180.000} C_DIS
LIN {X 85.276,Y 104.966,Z 69.000,A 180.000,B 0.000,C 180.000} C_DIS
LIN {X 85.368,Y 105.120,Z 69.000,A 180.000,B 0.000,C 180.000} C_DIS
LIN {X 85.455,Y 105.252,Z 69.000,A 180.000,B 0.000,C 180.000} C_DIS
LIN {X 85.725,Y 105.656,Z 69.000,A 180.000,B 0.000,C 180.000} C_DIS
LIN {X 85.813,Y 105.785,Z 69.000,A 180.000,B 0.000,C 180.000} C_DIS
LIN {X 85.849,Y 105.835,Z 69.000,A 180.000,B 0.000,C 180.000} C_DIS
LIN {X 85.983,Y 106.014,Z 69.000,A 180.000,B 0.000,C 180.000} C_DIS
LIN {X 86.252,Y 106.371,Z 69.000,A 180.000,B 0.000,C 180.000} C_DIS
LIN {X 86.349,Y 106.493,Z 69.000,A 180.000,B 0.000,C 180.000} C_DIS
LIN {X 86.707,Y 106.916,Z 69.000,A 180.000,B 0.000,C 180.000} C_DIS
LIN {X 86.855,Y 107.086,Z 69.000,A 180.000,B 0.000,C 180.000} C_DIS
LIN {X 86.885,Y 107.119,Z 69.000,A 180.000,B 0.000,C 180.000} C_DIS
LIN {X 87.243,Y 107.497,Z 69.000,A 180.000,B 0.000,C 180.000} C_DIS
LIN {X 87.363,Y 107.623,Z 69.000,A 180.000,B 0.000,C 180.000} C_DIS
LIN {X 87.422,Y 107.681,Z 69.000,A 180.000,B 0.000,C 180.000} C_DIS
LIN {X 87.779,Y 108.019,Z 69.000,A 180.000,B 0.000,C 180.000} C_DIS
LIN {X 87.928,Y 108.159,Z 69.000,A 180.000,B 0.000,C 180.000} C_DIS
LIN {X 87.958,Y 108.186,Z 69.000,A 180.000,B 0.000,C 180.000} C_DIS
LIN {X 88.137,Y 108.338,Z 69.000,A 180.000,B 0.000,C 180.000} C_DIS
LIN {X 88.494,Y 108.640,Z 69.000,A 180.000,B 0.000,C 180.000} C_DIS
LIN {X 88.562,Y 108.695,Z 69.000,A 180.000,B 0.000,C 180.000} C_DIS
LIN {X 88.673,Y 108.781,Z 69.000,A 180.000,B 0.000,C 180.000} C_DIS
LIN {X 89.034,Y 109.053,Z 69.000,A 180.000,B 0.000,C 180.000} C_DIS
LIN {X 89.209,Y 109.184,Z 69.000,A 180.000,B 0.000,C 180.000} C_DIS
LIN {X 89.280,Y 109.232,Z 69.000,A 180.000,B 0.000,C 180.000} C_DIS
LIN {X 89.746,Y 109.543,Z 69.000,A 180.000,B 0.000,C 180.000} C_DIS
LIN {X 89.815,Y 109.589,Z 69.000,A 180.000,B 0.000,C 180.000} C_DIS
LIN {X 89.925,Y 109.659,Z 69.000,A 180.000,B 0.000,C 180.000} C_DIS
LIN {X 90.110,Y 109.768,Z 69.000,A 180.000,B 0.000,C 180.000} C_DIS
LIN {X 90.461,Y 109.975,Z 69.000,A 180.000,B 0.000,C 180.000} C_DIS
LIN {X 90.640,Y 110.076,Z 69.000,A 180.000,B 0.000,C 180.000} C_DIS
LIN {X 91.176,Y 110.353,Z 69.000,A 180.000,B 0.000,C 180.000} C_DIS
LIN {X 91.355,Y 110.440,Z 69.000,A 180.000,B 0.000,C 180.000} C_DIS
LIN {X 91.561,Y 110.532,Z 69.000,A 180.000,B 0.000,C 180.000} C_DIS
; Link Move Starts
LIN {X 91.848,Y 110.661,Z 69.000,A 180.000,B 0.000,C 180.000} C_DIS
LIN {X 92.114,Y 110.774,Z 68.999,A 180.000,B 0.000,C 180.000} C_DIS
LIN {X 92.408,Y 110.887,Z 68.998,A 180.000,B 0.000,C 180.000} C_DIS
LIN {X 92.700,Y 110.999,Z 68.996,A 180.000,B 0.000,C 180.000} C_DIS
LIN {X 92.976,Y 111.092,Z 68.994,A 180.000,B 0.000,C 180.000} C_DIS
LIN {X 93.276,Y 111.189,Z 68.992,A 180.000,B 0.000,C 180.000} C_DIS
LIN {X 93.565,Y 111.280,Z 68.989,A 180.000,B 0.000,C 180.000} C_DIS
LIN {X 93.856,Y 111.357,Z 68.986,A 180.000,B 0.000,C 180.000} C_DIS
LIN {X 94.159,Y 111.437,Z 68.982,A 180.000,B 0.000,C 180.000} C_DIS
LIN {X 94.444,Y 111.504,Z 68.978,A 180.000,B 0.000,C 180.000} C_DIS
LIN {X 94.750,Y 111.568,Z 68.974,A 180.000,B 0.000,C 180.000} C_DIS
LIN {X 95.049,Y 111.629,Z 68.969,A 180.000,B 0.000,C 180.000} C_DIS
LIN {X 95.197,Y 111.654,Z 68.966,A 180.000,B 0.000,C 180.000} C_DIS
LIN {X 95.345,Y 111.676,Z 68.964,A 180.000,B 0.000,C 180.000} C_DIS
LIN {X 95.501,Y 111.700,Z 68.961,A 180.000,B 0.000,C 180.000} C_DIS
LIN {X 95.657,Y 111.723,Z 68.958,A 180.000,B 0.000,C 180.000} C_DIS
LIN {X 95.802,Y 111.745,Z 68.955,A 180.000,B 0.000,C 180.000} C_DIS
LIN {X 95.948,Y 111.764,Z 68.952,A 180.000,B 0.000,C 180.000} C_DIS
LIN {X 96.103,Y 111.778,Z 68.949,A 180.000,B 0.000,C 180.000} C_DIS
LIN {X 96.258,Y 111.793,Z 68.946,A 180.000,B 0.000,C 180.000} C_DIS
LIN {X 96.414,Y 111.808,Z 68.942,A 180.000,B 0.000,C 180.000} C_DIS
LIN {X 96.571,Y 111.822,Z 68.939,A 180.000,B 0.000,C 180.000} C_DIS
LIN {X 96.716,Y 111.834,Z 68.936,A 180.000,B 0.000,C 180.000} C_DIS
LIN {X 96.861,Y 111.841,Z 68.932,A 180.000,B 0.000,C 180.000} C_DIS
LIN {X 97.019,Y 111.847,Z 68.929,A 180.000,B 0.000,C 180.000} C_DIS
LIN {X 97.176,Y 111.853,Z 68.925,A 180.000,B 0.000,C 180.000} C_DIS
LIN {X 97.326,Y 111.859,Z 68.921,A 180.000,B 0.000,C 180.000} C_DIS
LIN {X 97.476,Y 111.865,Z 68.917,A 180.000,B 0.000,C 180.000} C_DIS
LIN {X 97.629,Y 111.864,Z 68.914,A 180.000,B 0.000,C 180.000} C_DIS
LIN {X 97.782,Y 111.861,Z 68.910,A 180.000,B 0.000,C 180.000} C_DIS
LIN {X 97.939,Y 111.859,Z 68.905,A 180.000,B 0.000,C 180.000} C_DIS
LIN {X 98.097,Y 111.856,Z 68.901,A 180.000,B 0.000,C 180.000} C_DIS
LIN {X 98.244,Y 111.854,Z 68.897,A 180.000,B 0.000,C 180.000} C_DIS
LIN {X 98.391,Y 111.847,Z 68.893,A 180.000,B 0.000,C 180.000} C_DIS
LIN {X 98.547,Y 111.836,Z 68.889,A 180.000,B 0.000,C 180.000} C_DIS
LIN {X 98.702,Y 111.825,Z 68.884,A 180.000,B 0.000,C 180.000} C_DIS
LIN {X 98.855,Y 111.814,Z 68.880,A 180.000,B 0.000,C 180.000} C_DIS
LIN {X 99.008,Y 111.803,Z 68.875,A 180.000,B 0.000,C 180.000} C_DIS
LIN {X 99.158,Y 111.790,Z 68.871,A 180.000,B 0.000,C 180.000} C_DIS
LIN {X 99.307,Y 111.772,Z 68.866,A 180.000,B 0.000,C 180.000} C_DIS
LIN {X 99.463,Y 111.752,Z 68.861,A 180.000,B 0.000,C 180.000} C_DIS
LIN {X 99.620,Y 111.732,Z 68.856,A 180.000,B 0.000,C 180.000} C_DIS
LIN {X 99.768,Y 111.713,Z 68.851,A 180.000,B 0.000,C 180.000} C_DIS
LIN {X 99.916,Y 111.693,Z 68.847,A 180.000,B 0.000,C 180.000} C_DIS
LIN {X 99.992,Y 111.680,Z 68.844,A 180.000,B 0.000,C 180.000} C_DIS
LIN {X 100.068,Y 111.666,Z 68.842,A 180.000,B 0.000,C 180.000} C_DIS
LIN {X 100.144,Y 111.652,Z 68.839,A 180.000,B 0.000,C 180.000} C_DIS
LIN {X 100.298,Y 111.624,Z 68.834,A 180.000,B 0.000,C 180.000} C_DIS
LIN {X 100.375,Y 111.610,Z 68.831,A 180.000,B 0.000,C 180.000} C_DIS
LIN {X 100.453,Y 111.596,Z 68.829,A 180.000,B 0.000,C 180.000} C_DIS
LIN {X 100.530,Y 111.582,Z 68.826,A 180.000,B 0.000,C 180.000} C_DIS
LIN {X 100.602,Y 111.569,Z 68.823,A 180.000,B 0.000,C 180.000} C_DIS
LIN {X 100.675,Y 111.555,Z 68.821,A 180.000,B 0.000,C 180.000} C_DIS
LIN {X 100.747,Y 111.540,Z 68.818,A 180.000,B 0.000,C 180.000} C_DIS
LIN {X 100.818,Y 111.523,Z 68.816,A 180.000,B 0.000,C 180.000} C_DIS
LIN {X 100.895,Y 111.505,Z 68.813,A 180.000,B 0.000,C 180.000} C_DIS
LIN {X 100.971,Y 111.486,Z 68.810,A 180.000,B 0.000,C 180.000} C_DIS
LIN {X 101.353,Y 111.394,Z 68.797,A 180.000,B 0.000,C 180.000} C_DIS
LIN {X 101.429,Y 111.376,Z 68.794,A 180.000,B 0.000,C 180.000} C_DIS
LIN {X 101.501,Y 111.357,Z 68.791,A 180.000,B 0.000,C 180.000} C_DIS
LIN {X 101.572,Y 111.337,Z 68.789,A 180.000,B 0.000,C 180.000} C_DIS
LIN {X 101.789,Y 111.271,Z 68.781,A 180.000,B 0.000,C 180.000} C_DIS
LIN {X 101.939,Y 111.226,Z 68.775,A 180.000,B 0.000,C 180.000} C_DIS
LIN {X 102.015,Y 111.203,Z 68.773,A 180.000,B 0.000,C 180.000} C_DIS
LIN {X 102.163,Y 111.159,Z 68.767,A 180.000,B 0.000,C 180.000} C_DIS
LIN {X 102.237,Y 111.136,Z 68.765,A 180.000,B 0.000,C 180.000} C_DIS
LIN {X 102.310,Y 111.112,Z 68.762,A 180.000,B 0.000,C 180.000} C_DIS
LIN {X 102.381,Y 111.086,Z 68.759,A 180.000,B 0.000,C 180.000} C_DIS
LIN {X 102.522,Y 111.035,Z 68.754,A 180.000,B 0.000,C 180.000} C_DIS
LIN {X 102.593,Y 111.009,Z 68.751,A 180.000,B 0.000,C 180.000} C_DIS
LIN {X 102.741,Y 110.956,Z 68.746,A 180.000,B 0.000,C 180.000} C_DIS
LIN {X 102.959,Y 110.876,Z 68.738,A 180.000,B 0.000,C 180.000} C_DIS
LIN {X 103.029,Y 110.850,Z 68.735,A 180.000,B 0.000,C 180.000} C_DIS
LIN {X 103.098,Y 110.822,Z 68.733,A 180.000,B 0.000,C 180.000} C_DIS
LIN {X 103.166,Y 110.792,Z 68.730,A 180.000,B 0.000,C 180.000} C_DIS
LIN {X 103.310,Y 110.731,Z 68.724,A 180.000,B 0.000,C 180.000} C_DIS
LIN {X 103.525,Y 110.638,Z 68.716,A 180.000,B 0.000,C 180.000} C_DIS
LIN {X 103.668,Y 110.577,Z 68.711,A 180.000,B 0.000,C 180.000} C_DIS
LIN {X 103.740,Y 110.546,Z 68.708,A 180.000,B 0.000,C 180.000} C_DIS
LIN {X 103.808,Y 110.515,Z 68.706,A 180.000,B 0.000,C 180.000} C_DIS
LIN {X 103.876,Y 110.482,Z 68.703,A 180.000,B 0.000,C 180.000} C_DIS
LIN {X 104.292,Y 110.275,Z 68.687,A 180.000,B 0.000,C 180.000} C_DIS
LIN {X 104.429,Y 110.207,Z 68.681,A 180.000,B 0.000,C 180.000} C_DIS
LIN {X 104.496,Y 110.173,Z 68.679,A 180.000,B 0.000,C 180.000} C_DIS
LIN {X 104.563,Y 110.136,Z 68.676,A 180.000,B 0.000,C 180.000} C_DIS
LIN {X 104.697,Y 110.060,Z 68.671,A 180.000,B 0.000,C 180.000} C_DIS
LIN {X 105.105,Y 109.829,Z 68.654,A 180.000,B 0.000,C 180.000} C_DIS
LIN {X 105.170,Y 109.792,Z 68.652,A 180.000,B 0.000,C 180.000} C_DIS
LIN {X 105.234,Y 109.753,Z 68.649,A 180.000,B 0.000,C 180.000} C_DIS
LIN {X 105.296,Y 109.713,Z 68.646,A 180.000,B 0.000,C 180.000} C_DIS
LIN {X 105.425,Y 109.630,Z 68.641,A 180.000,B 0.000,C 180.000} C_DIS
LIN {X 105.751,Y 109.420,Z 68.628,A 180.000,B 0.000,C 180.000} C_DIS
LIN {X 105.814,Y 109.379,Z 68.625,A 180.000,B 0.000,C 180.000} C_DIS
LIN {X 105.878,Y 109.338,Z 68.622,A 180.000,B 0.000,C 180.000} C_DIS
LIN {X 105.942,Y 109.293,Z 68.620,A 180.000,B 0.000,C 180.000} C_DIS
LIN {X 106.005,Y 109.247,Z 68.617,A 180.000,B 0.000,C 180.000} C_DIS
LIN {X 106.445,Y 108.927,Z 68.598,A 180.000,B 0.000,C 180.000} C_DIS
LIN {X 106.506,Y 108.882,Z 68.595,A 180.000,B 0.000,C 180.000} C_DIS
LIN {X 106.566,Y 108.837,Z 68.593,A 180.000,B 0.000,C 180.000} C_DIS
LIN {X 106.625,Y 108.789,Z 68.590,A 180.000,B 0.000,C 180.000} C_DIS
LIN {X 106.807,Y 108.640,Z 68.582,A 180.000,B 0.000,C 180.000} C_DIS
LIN {X 107.110,Y 108.393,Z 68.568,A 180.000,B 0.000,C 180.000} C_DIS
LIN {X 107.168,Y 108.345,Z 68.565,A 180.000,B 0.000,C 180.000} C_DIS
LIN {X 107.225,Y 108.295,Z 68.563,A 180.000,B 0.000,C 180.000} C_DIS
LIN {X 107.281,Y 108.244,Z 68.560,A 180.000,B 0.000,C 180.000} C_DIS
LIN {X 107.626,Y 107.928,Z 68.544,A 180.000,B 0.000,C 180.000} C_DIS
LIN {X 107.683,Y 107.876,Z 68.541,A 180.000,B 0.000,C 180.000} C_DIS
LIN {X 107.740,Y 107.824,Z 68.538,A 180.000,B 0.000,C 180.000} C_DIS
LIN {X 107.796,Y 107.771,Z 68.536,A 180.000,B 0.000,C 180.000} C_DIS
LIN {X 107.850,Y 107.716,Z 68.533,A 180.000,B 0.000,C 180.000} C_DIS
LIN {X 108.284,Y 107.271,Z 68.511,A 180.000,B 0.000,C 180.000} C_DIS
LIN {X 108.337,Y 107.217,Z 68.509,A 180.000,B 0.000,C 180.000} C_DIS
LIN {X 108.388,Y 107.161,Z 68.506,A 180.000,B 0.000,C 180.000} C_DIS
LIN {X 108.437,Y 107.105,Z 68.503,A 180.000,B 0.000,C 180.000} C_DIS
LIN {X 108.799,Y 106.689,Z 68.484,A 180.000,B 0.000,C 180.000} C_DIS
LIN {X 108.851,Y 106.630,Z 68.481,A 180.000,B 0.000,C 180.000} C_DIS
LIN {X 108.900,Y 106.572,Z 68.479,A 180.000,B 0.000,C 180.000} C_DIS
LIN {X 108.947,Y 106.513,Z 68.476,A 180.000,B 0.000,C 180.000} C_DIS
LIN {X 109.328,Y 106.023,Z 68.454,A 180.000,B 0.000,C 180.000} C_DIS
LIN {X 109.375,Y 105.962,Z 68.452,A 180.000,B 0.000,C 180.000} C_DIS
LIN {X 109.420,Y 105.901,Z 68.449,A 180.000,B 0.000,C 180.000} C_DIS
LIN {X 109.464,Y 105.837,Z 68.446,A 180.000,B 0.000,C 180.000} C_DIS
LIN {X 109.820,Y 105.323,Z 68.425,A 180.000,B 0.000,C 180.000} C_DIS
LIN {X 109.862,Y 105.260,Z 68.422,A 180.000,B 0.000,C 180.000} C_DIS
LIN {X 109.902,Y 105.196,Z 68.419,A 180.000,B 0.000,C 180.000} C_DIS
LIN {X 110.024,Y 104.996,Z 68.411,A 180.000,B 0.000,C 180.000} C_DIS
LIN {X 110.228,Y 104.663,Z 68.397,A 180.000,B 0.000,C 180.000} C_DIS
LIN {X 110.269,Y 104.596,Z 68.395,A 180.000,B 0.000,C 180.000} C_DIS
LIN {X 110.307,Y 104.529,Z 68.392,A 180.000,B 0.000,C 180.000} C_DIS
LIN {X 110.344,Y 104.462,Z 68.389,A 180.000,B 0.000,C 180.000} C_DIS
LIN {X 110.638,Y 103.913,Z 68.368,A 180.000,B 0.000,C 180.000} C_DIS
LIN {X 110.674,Y 103.846,Z 68.365,A 180.000,B 0.000,C 180.000} C_DIS
LIN {X 110.707,Y 103.777,Z 68.362,A 180.000,B 0.000,C 180.000} C_DIS
LIN {X 110.807,Y 103.563,Z 68.354,A 180.000,B 0.000,C 180.000} C_DIS
LIN {X 110.873,Y 103.420,Z 68.349,A 180.000,B 0.000,C 180.000} C_DIS
LIN {X 110.940,Y 103.278,Z 68.343,A 180.000,B 0.000,C 180.000} C_DIS
LIN {X 110.973,Y 103.207,Z 68.340,A 180.000,B 0.000,C 180.000} C_DIS
LIN {X 111.005,Y 103.137,Z 68.338,A 180.000,B 0.000,C 180.000} C_DIS
LIN {X 111.036,Y 103.067,Z 68.335,A 180.000,B 0.000,C 180.000} C_DIS
LIN {X 111.065,Y 102.996,Z 68.332,A 180.000,B 0.000,C 180.000} C_DIS
LIN {X 111.093,Y 102.924,Z 68.330,A 180.000,B 0.000,C 180.000} C_DIS
LIN {X 111.152,Y 102.778,Z 68.324,A 180.000,B 0.000,C 180.000} C_DIS
LIN {X 111.297,Y 102.416,Z 68.311,A 180.000,B 0.000,C 180.000} C_DIS
LIN {X 111.325,Y 102.344,Z 68.308,A 180.000,B 0.000,C 180.000} C_DIS
LIN {X 111.351,Y 102.271,Z 68.305,A 180.000,B 0.000,C 180.000} C_DIS
LIN {X 111.401,Y 102.123,Z 68.300,A 180.000,B 0.000,C 180.000} C_DIS
LIN {X 111.426,Y 102.048,Z 68.297,A 180.000,B 0.000,C 180.000} C_DIS
LIN {X 111.476,Y 101.899,Z 68.291,A 180.000,B 0.000,C 180.000} C_DIS
LIN {X 111.551,Y 101.677,Z 68.283,A 180.000,B 0.000,C 180.000} C_DIS
LIN {X 111.575,Y 101.604,Z 68.281,A 180.000,B 0.000,C 180.000} C_DIS
LIN {X 111.598,Y 101.530,Z 68.278,A 180.000,B 0.000,C 180.000} C_DIS
LIN {X 111.619,Y 101.456,Z 68.275,A 180.000,B 0.000,C 180.000} C_DIS
LIN {X 111.660,Y 101.304,Z 68.270,A 180.000,B 0.000,C 180.000} C_DIS
LIN {X 111.723,Y 101.077,Z 68.261,A 180.000,B 0.000,C 180.000} C_DIS
LIN {X 111.765,Y 100.925,Z 68.256,A 180.000,B 0.000,C 180.000} C_DIS
LIN {X 111.786,Y 100.849,Z 68.253,A 180.000,B 0.000,C 180.000} C_DIS
LIN {X 111.806,Y 100.774,Z 68.250,A 180.000,B 0.000,C 180.000} C_DIS
LIN {X 111.823,Y 100.699,Z 68.248,A 180.000,B 0.000,C 180.000} C_DIS
LIN {X 111.872,Y 100.471,Z 68.240,A 180.000,B 0.000,C 180.000} C_DIS
LIN {X 111.906,Y 100.317,Z 68.234,A 180.000,B 0.000,C 180.000} C_DIS
LIN {X 111.922,Y 100.240,Z 68.231,A 180.000,B 0.000,C 180.000} C_DIS
LIN {X 111.955,Y 100.087,Z 68.226,A 180.000,B 0.000,C 180.000} C_DIS
LIN {X 111.972,Y 100.011,Z 68.223,A 180.000,B 0.000,C 180.000} C_DIS
LIN {X 111.987,Y 99.934,Z 68.220,A 180.000,B 0.000,C 180.000} C_DIS
LIN {X 111.999,Y 99.857,Z 68.218,A 180.000,B 0.000,C 180.000} C_DIS
LIN {X 112.023,Y 99.703,Z 68.212,A 180.000,B 0.000,C 180.000} C_DIS
LIN {X 112.035,Y 99.627,Z 68.210,A 180.000,B 0.000,C 180.000} C_DIS
LIN {X 112.060,Y 99.471,Z 68.204,A 180.000,B 0.000,C 180.000} C_DIS
LIN {X 112.097,Y 99.239,Z 68.196,A 180.000,B 0.000,C 180.000} C_DIS
LIN {X 112.108,Y 99.162,Z 68.193,A 180.000,B 0.000,C 180.000} C_DIS
LIN {X 112.117,Y 99.085,Z 68.190,A 180.000,B 0.000,C 180.000} C_DIS
LIN {X 112.125,Y 99.008,Z 68.188,A 180.000,B 0.000,C 180.000} C_DIS
LIN {X 112.133,Y 98.930,Z 68.185,A 180.000,B 0.000,C 180.000} C_DIS
LIN {X 112.141,Y 98.851,Z 68.182,A 180.000,B 0.000,C 180.000} C_DIS
LIN {X 112.149,Y 98.773,Z 68.180,A 180.000,B 0.000,C 180.000} C_DIS
LIN {X 112.157,Y 98.695,Z 68.177,A 180.000,B 0.000,C 180.000} C_DIS
LIN {X 112.164,Y 98.616,Z 68.174,A 180.000,B 0.000,C 180.000} C_DIS
LIN {X 112.172,Y 98.538,Z 68.172,A 180.000,B 0.000,C 180.000} C_DIS
LIN {X 112.180,Y 98.460,Z 68.169,A 180.000,B 0.000,C 180.000} C_DIS
LIN {X 112.188,Y 98.382,Z 68.166,A 180.000,B 0.000,C 180.000} C_DIS
LIN {X 112.194,Y 98.304,Z 68.164,A 180.000,B 0.000,C 180.000} C_DIS
LIN {X 112.198,Y 98.226,Z 68.161,A 180.000,B 0.000,C 180.000} C_DIS
LIN {X 112.201,Y 98.149,Z 68.159,A 180.000,B 0.000,C 180.000} C_DIS
LIN {X 112.211,Y 97.914,Z 68.151,A 180.000,B 0.000,C 180.000} C_DIS
LIN {X 112.215,Y 97.835,Z 68.149,A 180.000,B 0.000,C 180.000} C_DIS
LIN {X 112.218,Y 97.756,Z 68.146,A 180.000,B 0.000,C 180.000} C_DIS
LIN {X 112.225,Y 97.599,Z 68.141,A 180.000,B 0.000,C 180.000} C_DIS
LIN {X 112.228,Y 97.443,Z 68.136,A 180.000,B 0.000,C 180.000} C_DIS
LIN {X 112.226,Y 97.286,Z 68.132,A 180.000,B 0.000,C 180.000} C_DIS
LIN {X 112.224,Y 97.130,Z 68.127,A 180.000,B 0.000,C 180.000} C_DIS
LIN {X 112.222,Y 96.972,Z 68.122,A 180.000,B 0.000,C 180.000} C_DIS
LIN {X 112.219,Y 96.815,Z 68.118,A 180.000,B 0.000,C 180.000} C_DIS
LIN {X 112.216,Y 96.659,Z 68.113,A 180.000,B 0.000,C 180.000} C_DIS
LIN {X 112.205,Y 96.503,Z 68.109,A 180.000,B 0.000,C 180.000} C_DIS
LIN {X 112.194,Y 96.346,Z 68.104,A 180.000,B 0.000,C 180.000} C_DIS
LIN {X 112.183,Y 96.189,Z 68.100,A 180.000,B 0.000,C 180.000} C_DIS
LIN {X 112.172,Y 96.032,Z 68.096,A 180.000,B 0.000,C 180.000} C_DIS
LIN {X 112.160,Y 95.875,Z 68.092,A 180.000,B 0.000,C 180.000} C_DIS
LIN {X 112.142,Y 95.720,Z 68.088,A 180.000,B 0.000,C 180.000} C_DIS
LIN {X 112.122,Y 95.564,Z 68.084,A 180.000,B 0.000,C 180.000} C_DIS
LIN {X 112.101,Y 95.408,Z 68.080,A 180.000,B 0.000,C 180.000} C_DIS
LIN {X 112.081,Y 95.252,Z 68.076,A 180.000,B 0.000,C 180.000} C_DIS
LIN {X 112.061,Y 95.096,Z 68.072,A 180.000,B 0.000,C 180.000} C_DIS
LIN {X 112.036,Y 94.941,Z 68.068,A 180.000,B 0.000,C 180.000} C_DIS
LIN {X 112.007,Y 94.787,Z 68.065,A 180.000,B 0.000,C 180.000} C_DIS
LIN {X 111.978,Y 94.633,Z 68.061,A 180.000,B 0.000,C 180.000} C_DIS
LIN {X 111.949,Y 94.478,Z 68.058,A 180.000,B 0.000,C 180.000} C_DIS
LIN {X 111.920,Y 94.323,Z 68.054,A 180.000,B 0.000,C 180.000} C_DIS
LIN {X 111.888,Y 94.169,Z 68.051,A 180.000,B 0.000,C 180.000} C_DIS
LIN {X 111.850,Y 94.017,Z 68.048,A 180.000,B 0.000,C 180.000} C_DIS
LIN {X 111.812,Y 93.864,Z 68.045,A 180.000,B 0.000,C 180.000} C_DIS
LIN {X 111.774,Y 93.711,Z 68.042,A 180.000,B 0.000,C 180.000} C_DIS
LIN {X 111.736,Y 93.559,Z 68.039,A 180.000,B 0.000,C 180.000} C_DIS
LIN {X 111.697,Y 93.406,Z 68.036,A 180.000,B 0.000,C 180.000} C_DIS
LIN {X 111.651,Y 93.256,Z 68.034,A 180.000,B 0.000,C 180.000} C_DIS
LIN {X 111.605,Y 93.106,Z 68.031,A 180.000,B 0.000,C 180.000} C_DIS
LIN {X 111.511,Y 92.805,Z 68.026,A 180.000,B 0.000,C 180.000} C_DIS
LIN {X 111.412,Y 92.507,Z 68.022,A 180.000,B 0.000,C 180.000} C_DIS
LIN {X 111.301,Y 92.212,Z 68.017,A 180.000,B 0.000,C 180.000} C_DIS
LIN {X 111.190,Y 91.917,Z 68.014,A 180.000,B 0.000,C 180.000} C_DIS
LIN {X 111.067,Y 91.627,Z 68.010,A 180.000,B 0.000,C 180.000} C_DIS
LIN {X 110.940,Y 91.339,Z 68.008,A 180.000,B 0.000,C 180.000} C_DIS
LIN {X 110.810,Y 91.052,Z 68.005,A 180.000,B 0.000,C 180.000} C_DIS
LIN {X 110.667,Y 90.772,Z 68.003,A 180.000,B 0.000,C 180.000} C_DIS
LIN {X 110.523,Y 90.492,Z 68.002,A 180.000,B 0.000,C 180.000} C_DIS
LIN {X 110.371,Y 90.216,Z 68.001,A 180.000,B 0.000,C 180.000} C_DIS
LIN {X 110.212,Y 89.944,Z 68.000,A 180.000,B 0.000,C 180.000} C_DIS
LIN {X 110.113,Y 89.778,Z 68.000,A 180.000,B 0.000,C 180.000} C_DIS
; Cutting Move Starts
LIN {X 110.094,Y 89.746,Z 68.000,A 180.000,B 0.000,C 180.000} C_DIS
LIN {X 109.983,Y 89.567,Z 68.000,A 180.000,B 0.000,C 180.000} C_DIS
LIN {X 109.625,Y 89.031,Z 68.000,A 180.000,B 0.000,C 180.000} C_DIS
LIN {X 109.589,Y 88.977,Z 68.000,A 180.000,B 0.000,C 180.000} C_DIS
LIN {X 109.498,Y 88.852,Z 68.000,A 180.000,B 0.000,C 180.000} C_DIS
LIN {X 109.229,Y 88.494,Z 68.000,A 180.000,B 0.000,C 180.000} C_DIS
LIN {X 109.094,Y 88.316,Z 68.000,A 180.000,B 0.000,C 180.000} C_DIS
LIN {X 109.053,Y 88.263,Z 68.000,A 180.000,B 0.000,C 180.000} C_DIS
LIN {X 108.947,Y 88.137,Z 68.000,A 180.000,B 0.000,C 180.000} C_DIS
LIN {X 108.645,Y 87.779,Z 68.000,A 180.000,B 0.000,C 180.000} C_DIS
LIN {X 108.517,Y 87.629,Z 68.000,A 180.000,B 0.000,C 180.000} C_DIS
LIN {X 108.490,Y 87.601,Z 68.000,A 180.000,B 0.000,C 180.000} C_DIS
LIN {X 108.321,Y 87.422,Z 68.000,A 180.000,B 0.000,C 180.000} C_DIS
LIN {X 108.152,Y 87.243,Z 68.000,A 180.000,B 0.000,C 180.000} C_DIS
LIN {X 107.983,Y 87.064,Z 68.000,A 180.000,B 0.000,C 180.000} C_DIS
LIN {X 107.980,Y 87.062,Z 68.000,A 180.000,B 0.000,C 180.000} C_DIS
LIN {X 107.802,Y 86.890,Z 68.000,A 180.000,B 0.000,C 180.000} C_DIS
LIN {X 107.419,Y 86.528,Z 68.000,A 180.000,B 0.000,C 180.000} C_DIS
LIN {X 107.265,Y 86.392,Z 68.000,A 180.000,B 0.000,C 180.000} C_DIS
LIN {X 106.791,Y 85.992,Z 68.000,A 180.000,B 0.000,C 180.000} C_DIS
LIN {X 106.729,Y 85.940,Z 68.000,A 180.000,B 0.000,C 180.000} C_DIS
LIN {X 106.561,Y 85.813,Z 68.000,A 180.000,B 0.000,C 180.000} C_DIS
LIN {X 106.193,Y 85.535,Z 68.000,A 180.000,B 0.000,C 180.000} C_DIS
LIN {X 106.086,Y 85.455,Z 68.000,A 180.000,B 0.000,C 180.000} C_DIS
LIN {X 106.014,Y 85.405,Z 68.000,A 180.000,B 0.000,C 180.000} C_DIS
LIN {X 105.822,Y 85.276,Z 68.000,A 180.000,B 0.000,C 180.000} C_DIS
LIN {X 105.477,Y 85.046,Z 68.000,A 180.000,B 0.000,C 180.000} C_DIS
LIN {X 105.299,Y 84.932,Z 68.000,A 180.000,B 0.000,C 180.000} C_DIS
LIN {X 104.762,Y 84.616,Z 68.000,A 180.000,B 0.000,C 180.000} C_DIS
LIN {X 104.669,Y 84.561,Z 68.000,A 180.000,B 0.000,C 180.000} C_DIS
LIN {X 104.584,Y 84.516,Z 68.000,A 180.000,B 0.000,C 180.000} C_DIS
LIN {X 103.980,Y 84.204,Z 68.000,A 180.000,B 0.000,C 180.000} C_DIS
LIN {X 103.869,Y 84.150,Z 68.000,A 180.000,B 0.000,C 180.000} C_DIS
LIN {X 103.690,Y 84.070,Z 68.000,A 180.000,B 0.000,C 180.000} C_DIS
LIN {X 103.332,Y 83.910,Z 68.000,A 180.000,B 0.000,C 180.000} C_DIS
LIN {X 103.189,Y 83.846,Z 68.000,A 180.000,B 0.000,C 180.000} C_DIS
LIN {X 103.153,Y 83.831,Z 68.000,A 180.000,B 0.000,C 180.000} C_DIS
LIN {X 102.975,Y 83.762,Z 68.000,A 180.000,B 0.000,C 180.000} C_DIS
LIN {X 102.617,Y 83.626,Z 68.000,A 180.000,B 0.000,C 180.000} C_DIS
LIN {X 102.438,Y 83.557,Z 68.000,A 180.000,B 0.000,C 180.000} C_DIS
LIN {X 102.260,Y 83.497,Z 68.000,A 180.000,B 0.000,C 180.000} C_DIS
LIN {X 101.672,Y 83.310,Z 68.000,A 180.000,B 0.000,C 180.000} C_DIS
LIN {X 101.545,Y 83.272,Z 68.000,A 180.000,B 0.000,C 180.000} C_DIS
LIN {X 101.366,Y 83.226,Z 68.000,A 180.000,B 0.000,C 180.000} C_DIS
LIN {X 100.998,Y 83.131,Z 68.000,A 180.000,B 0.000,C 180.000} C_DIS
LIN {X 100.829,Y 83.088,Z 68.000,A 180.000,B 0.000,C 180.000} C_DIS
LIN {X 100.651,Y 83.050,Z 68.000,A 180.000,B 0.000,C 180.000} C_DIS
LIN {X 100.114,Y 82.943,Z 68.000,A 180.000,B 0.000,C 180.000} C_DIS
LIN {X 99.936,Y 82.910,Z 68.000,A 180.000,B 0.000,C 180.000} C_DIS
LIN {X 99.757,Y 82.885,Z 68.000,A 180.000,B 0.000,C 180.000} C_DIS
LIN {X 99.221,Y 82.809,Z 68.000,A 180.000,B 0.000,C 180.000} C_DIS
LIN {X 99.042,Y 82.791,Z 68.000,A 180.000,B 0.000,C 180.000} C_DIS
LIN {X 98.505,Y 82.745,Z 68.000,A 180.000,B 0.000,C 180.000} C_DIS
LIN {X 98.327,Y 82.731,Z 68.000,A 180.000,B 0.000,C 180.000} C_DIS
LIN {X 98.148,Y 82.725,Z 68.000,A 180.000,B 0.000,C 180.000} C_DIS
LIN {X 97.612,Y 82.710,Z 68.000,A 180.000,B 0.000,C 180.000} C_DIS
LIN {X 97.433,Y 82.709,Z 68.000,A 180.000,B 0.000,C 180.000} C_DIS
LIN {X 96.897,Y 82.724,Z 68.000,A 180.000,B 0.000,C 180.000} C_DIS
LIN {X 96.718,Y 82.729,Z 68.000,A 180.000,B 0.000,C 180.000} C_DIS
LIN {X 96.539,Y 82.742,Z 68.000,A 180.000,B 0.000,C 180.000} C_DIS
LIN {X 96.003,Y 82.787,Z 68.000,A 180.000,B 0.000,C 180.000} C_DIS
LIN {X 95.824,Y 82.804,Z 68.000,A 180.000,B 0.000,C 180.000} C_DIS
LIN {X 95.645,Y 82.828,Z 68.000,A 180.000,B 0.000,C 180.000} C_DIS
LIN {X 95.109,Y 82.904,Z 68.000,A 180.000,B 0.000,C 180.000} C_DIS
LIN {X 94.930,Y 82.935,Z 68.000,A 180.000,B 0.000,C 180.000} C_DIS
LIN {X 94.394,Y 83.041,Z 68.000,A 180.000,B 0.000,C 180.000} C_DIS
LIN {X 94.215,Y 83.078,Z 68.000,A 180.000,B 0.000,C 180.000} C_DIS
LIN {X 94.036,Y 83.122,Z 68.000,A 180.000,B 0.000,C 180.000} C_DIS
LIN {X 93.500,Y 83.261,Z 68.000,A 180.000,B 0.000,C 180.000} C_DIS
LIN {X 93.328,Y 83.310,Z 68.000,A 180.000,B 0.000,C 180.000} C_DIS
LIN {X 92.767,Y 83.489,Z 68.000,A 180.000,B 0.000,C 180.000} C_DIS
LIN {X 92.606,Y 83.541,Z 68.000,A 180.000,B 0.000,C 180.000} C_DIS
LIN {X 92.427,Y 83.609,Z 68.000,A 180.000,B 0.000,C 180.000} C_DIS
LIN {X 92.070,Y 83.745,Z 68.000,A 180.000,B 0.000,C 180.000} C_DIS
LIN {X 91.891,Y 83.813,Z 68.000,A 180.000,B 0.000,C 180.000} C_DIS
LIN {X 91.811,Y 83.846,Z 68.000,A 180.000,B 0.000,C 180.000} C_DIS
LIN {X 91.712,Y 83.890,Z 68.000,A 180.000,B 0.000,C 180.000} C_DIS
LIN {X 91.176,Y 84.130,Z 68.000,A 180.000,B 0.000,C 180.000} C_DIS
LIN {X 91.020,Y 84.204,Z 68.000,A 180.000,B 0.000,C 180.000} C_DIS
LIN {X 90.461,Y 84.493,Z 68.000,A 180.000,B 0.000,C 180.000} C_DIS
LIN {X 90.331,Y 84.561,Z 68.000,A 180.000,B 0.000,C 180.000} C_DIS
LIN {X 90.282,Y 84.590,Z 68.000,A 180.000,B 0.000,C 180.000} C_DIS
LIN {X 89.724,Y 84.919,Z 68.000,A 180.000,B 0.000,C 180.000} C_DIS
LIN {X 89.567,Y 85.017,Z 68.000,A 180.000,B 0.000,C 180.000} C_DIS
LIN {X 89.031,Y 85.375,Z 68.000,A 180.000,B 0.000,C 180.000} C_DIS
LIN {X 88.914,Y 85.455,Z 68.000,A 180.000,B 0.000,C 180.000} C_DIS
LIN {X 88.852,Y 85.502,Z 68.000,A 180.000,B 0.000,C 180.000} C_DIS
LIN {X 88.439,Y 85.813,Z 68.000,A 180.000,B 0.000,C 180.000} C_DIS
LIN {X 88.316,Y 85.906,Z 68.000,A 180.000,B 0.000,C 180.000} C_DIS
LIN {X 88.209,Y 85.992,Z 68.000,A 180.000,B 0.000,C 180.000} C_DIS
LIN {X 87.779,Y 86.355,Z 68.000,A 180.000,B 0.000,C 180.000} C_DIS
LIN {X 87.601,Y 86.510,Z 68.000,A 180.000,B 0.000,C 180.000} C_DIS
LIN {X 87.581,Y 86.528,Z 68.000,A 180.000,B 0.000,C 180.000} C_DIS
LIN {X 87.203,Y 86.885,Z 68.000,A 180.000,B 0.000,C 180.000} C_DIS
LIN {X 87.064,Y 87.017,Z 68.000,A 180.000,B 0.000,C 180.000} C_DIS
LIN {X 87.017,Y 87.064,Z 68.000,A 180.000,B 0.000,C 180.000} C_DIS
LIN {X 86.885,Y 87.203,Z 68.000,A 180.000,B 0.000,C 180.000} C_DIS
LIN {X 86.528,Y 87.582,Z 68.000,A 180.000,B 0.000,C 180.000} C_DIS
LIN {X 86.510,Y 87.601,Z 68.000,A 180.000,B 0.000,C 180.000} C_DIS
LIN {X 86.355,Y 87.779,Z 68.000,A 180.000,B 0.000,C 180.000} C_DIS
LIN {X 85.992,Y 88.209,Z 68.000,A 180.000,B 0.000,C 180.000} C_DIS
LIN {X 85.906,Y 88.316,Z 68.000,A 180.000,B 0.000,C 180.000} C_DIS
LIN {X 85.813,Y 88.439,Z 68.000,A 180.000,B 0.000,C 180.000} C_DIS
LIN {X 85.502,Y 88.852,Z 68.000,A 180.000,B 0.000,C 180.000} C_DIS
LIN {X 85.455,Y 88.914,Z 68.000,A 180.000,B 0.000,C 180.000} C_DIS
LIN {X 85.375,Y 89.031,Z 68.000,A 180.000,B 0.000,C 180.000} C_DIS
LIN {X 85.017,Y 89.567,Z 68.000,A 180.000,B 0.000,C 180.000} C_DIS
LIN {X 84.919,Y 89.724,Z 68.000,A 180.000,B 0.000,C 180.000} C_DIS
LIN {X 84.590,Y 90.282,Z 68.000,A 180.000,B 0.000,C 180.000} C_DIS
LIN {X 84.561,Y 90.332,Z 68.000,A 180.000,B 0.000,C 180.000} C_DIS
LIN {X 84.493,Y 90.461,Z 68.000,A 180.000,B 0.000,C 180.000} C_DIS
LIN {X 84.204,Y 91.020,Z 68.000,A 180.000,B 0.000,C 180.000} C_DIS
LIN {X 84.130,Y 91.176,Z 68.000,A 180.000,B 0.000,C 180.000} C_DIS
LIN {X 83.890,Y 91.712,Z 68.000,A 180.000,B 0.000,C 180.000} C_DIS
LIN {X 83.846,Y 91.811,Z 68.000,A 180.000,B 0.000,C 180.000} C_DIS
LIN {X 83.814,Y 91.891,Z 68.000,A 180.000,B 0.000,C 180.000} C_DIS
LIN {X 83.745,Y 92.070,Z 68.000,A 180.000,B 0.000,C 180.000} C_DIS
LIN {X 83.609,Y 92.427,Z 68.000,A 180.000,B 0.000,C 180.000} C_DIS
LIN {X 83.541,Y 92.606,Z 68.000,A 180.000,B 0.000,C 180.000} C_DIS
LIN {X 83.489,Y 92.766,Z 68.000,A 180.000,B 0.000,C 180.000} C_DIS
LIN {X 83.310,Y 93.327,Z 68.000,A 180.000,B 0.000,C 180.000} C_DIS
LIN {X 83.261,Y 93.500,Z 68.000,A 180.000,B 0.000,C 180.000} C_DIS
LIN {X 83.123,Y 94.036,Z 68.000,A 180.000,B 0.000,C 180.000} C_DIS
LIN {X 83.078,Y 94.215,Z 68.000,A 180.000,B 0.000,C 180.000} C_DIS
LIN {X 83.041,Y 94.394,Z 68.000,A 180.000,B 0.000,C 180.000} C_DIS
LIN {X 82.935,Y 94.930,Z 68.000,A 180.000,B 0.000,C 180.000} C_DIS
LIN {X 82.904,Y 95.109,Z 68.000,A 180.000,B 0.000,C 180.000} C_DIS
LIN {X 82.828,Y 95.645,Z 68.000,A 180.000,B 0.000,C 180.000} C_DIS
LIN {X 82.815,Y 95.740,Z 68.000,A 180.000,B 0.000,C 180.000} C_DIS
LIN {X 82.804,Y 95.824,Z 68.000,A 180.000,B 0.000,C 180.000} C_DIS
LIN {X 82.787,Y 96.003,Z 68.000,A 180.000,B 0.000,C 180.000} C_DIS
LIN {X 82.742,Y 96.539,Z 68.000,A 180.000,B 0.000,C 180.000} C_DIS
LIN {X 82.729,Y 96.718,Z 68.000,A 180.000,B 0.000,C 180.000} C_DIS
LIN {X 82.724,Y 96.897,Z 68.000,A 180.000,B 0.000,C 180.000} C_DIS
LIN {X 82.714,Y 97.254,Z 68.000,A 180.000,B 0.000,C 180.000} C_DIS
LIN {X 82.709,Y 97.433,Z 68.000,A 180.000,B 0.000,C 180.000} C_DIS
LIN {X 82.710,Y 97.612,Z 68.000,A 180.000,B 0.000,C 180.000} C_DIS
LIN {X 82.725,Y 98.148,Z 68.000,A 180.000,B 0.000,C 180.000} C_DIS
LIN {X 82.731,Y 98.327,Z 68.000,A 180.000,B 0.000,C 180.000} C_DIS
LIN {X 82.745,Y 98.505,Z 68.000,A 180.000,B 0.000,C 180.000} C_DIS
LIN {X 82.791,Y 99.042,Z 68.000,A 180.000,B 0.000,C 180.000} C_DIS
LIN {X 82.809,Y 99.221,Z 68.000,A 180.000,B 0.000,C 180.000} C_DIS
LIN {X 82.835,Y 99.399,Z 68.000,A 180.000,B 0.000,C 180.000} C_DIS
LIN {X 82.885,Y 99.757,Z 68.000,A 180.000,B 0.000,C 180.000} C_DIS
LIN {X 82.910,Y 99.936,Z 68.000,A 180.000,B 0.000,C 180.000} C_DIS
LIN {X 82.943,Y 100.114,Z 68.000,A 180.000,B 0.000,C 180.000} C_DIS
LIN {X 83.050,Y 100.651,Z 68.000,A 180.000,B 0.000,C 180.000} C_DIS
LIN {X 83.088,Y 100.829,Z 68.000,A 180.000,B 0.000,C 180.000} C_DIS
LIN {X 83.131,Y 100.997,Z 68.000,A 180.000,B 0.000,C 180.000} C_DIS
LIN {X 83.226,Y 101.366,Z 68.000,A 180.000,B 0.000,C 180.000} C_DIS
LIN {X 83.272,Y 101.545,Z 68.000,A 180.000,B 0.000,C 180.000} C_DIS
LIN {X 83.310,Y 101.673,Z 68.000,A 180.000,B 0.000,C 180.000} C_DIS
LIN {X 83.497,Y 102.260,Z 68.000,A 180.000,B 0.000,C 180.000} C_DIS
LIN {X 83.558,Y 102.438,Z 68.000,A 180.000,B 0.000,C 180.000} C_DIS
LIN {X 83.626,Y 102.617,Z 68.000,A 180.000,B 0.000,C 180.000} C_DIS
LIN {X 83.762,Y 102.975,Z 68.000,A 180.000,B 0.000,C 180.000} C_DIS
LIN {X 83.831,Y 103.153,Z 68.000,A 180.000,B 0.000,C 180.000} C_DIS
LIN {X 83.846,Y 103.189,Z 68.000,A 180.000,B 0.000,C 180.000} C_DIS
LIN {X 83.910,Y 103.332,Z 68.000,A 180.000,B 0.000,C 180.000} C_DIS
LIN {X 84.070,Y 103.690,Z 68.000,A 180.000,B 0.000,C 180.000} C_DIS
LIN {X 84.150,Y 103.869,Z 68.000,A 180.000,B 0.000,C 180.000} C_DIS
LIN {X 84.204,Y 103.980,Z 68.000,A 180.000,B 0.000,C 180.000} C_DIS
LIN {X 84.516,Y 104.584,Z 68.000,A 180.000,B 0.000,C 180.000} C_DIS
LIN {X 84.561,Y 104.668,Z 68.000,A 180.000,B 0.000,C 180.000} C_DIS
LIN {X 84.616,Y 104.762,Z 68.000,A 180.000,B 0.000,C 180.000} C_DIS
LIN {X 84.932,Y 105.299,Z 68.000,A 180.000,B 0.000,C 180.000} C_DIS
LIN {X 85.046,Y 105.477,Z 68.000,A 180.000,B 0.000,C 180.000} C_DIS
LIN {X 85.285,Y 105.835,Z 68.000,A 180.000,B 0.000,C 180.000} C_DIS
LIN {X 85.405,Y 106.014,Z 68.000,A 180.000,B 0.000,C 180.000} C_DIS
LIN {X 85.455,Y 106.086,Z 68.000,A 180.000,B 0.000,C 180.000} C_DIS
LIN {X 85.535,Y 106.193,Z 68.000,A 180.000,B 0.000,C 180.000} C_DIS
LIN {X 85.813,Y 106.561,Z 68.000,A 180.000,B 0.000,C 180.000} C_DIS
LIN {X 85.940,Y 106.729,Z 68.000,A 180.000,B 0.000,C 180.000} C_DIS
LIN {X 85.992,Y 106.791,Z 68.000,A 180.000,B 0.000,C 180.000} C_DIS
LIN {X 86.392,Y 107.265,Z 68.000,A 180.000,B 0.000,C 180.000} C_DIS
LIN {X 86.528,Y 107.418,Z 68.000,A 180.000,B 0.000,C 180.000} C_DIS
LIN {X 86.890,Y 107.802,Z 68.000,A 180.000,B 0.000,C 180.000} C_DIS
LIN {X 87.062,Y 107.980,Z 68.000,A 180.000,B 0.000,C 180.000} C_DIS
LIN {X 87.064,Y 107.983,Z 68.000,A 180.000,B 0.000,C 180.000} C_DIS
LIN {X 87.243,Y 108.152,Z 68.000,A 180.000,B 0.000,C 180.000} C_DIS
LIN {X 87.439,Y 108.338,Z 68.000,A 180.000,B 0.000,C 180.000} C_DIS
LIN {X 87.601,Y 108.490,Z 68.000,A 180.000,B 0.000,C 180.000} C_DIS
LIN {X 87.629,Y 108.517,Z 68.000,A 180.000,B 0.000,C 180.000} C_DIS
LIN {X 87.779,Y 108.645,Z 68.000,A 180.000,B 0.000,C 180.000} C_DIS
LIN {X 88.137,Y 108.947,Z 68.000,A 180.000,B 0.000,C 180.000} C_DIS
LIN {X 88.263,Y 109.053,Z 68.000,A 180.000,B 0.000,C 180.000} C_DIS
LIN {X 88.316,Y 109.094,Z 68.000,A 180.000,B 0.000,C 180.000} C_DIS
LIN {X 88.498,Y 109.232,Z 68.000,A 180.000,B 0.000,C 180.000} C_DIS
LIN {X 88.852,Y 109.498,Z 68.000,A 180.000,B 0.000,C 180.000} C_DIS
LIN {X 88.977,Y 109.589,Z 68.000,A 180.000,B 0.000,C 180.000} C_DIS
LIN {X 89.031,Y 109.625,Z 68.000,A 180.000,B 0.000,C 180.000} C_DIS
LIN {X 89.567,Y 109.983,Z 68.000,A 180.000,B 0.000,C 180.000} C_DIS
LIN {X 89.746,Y 110.094,Z 68.000,A 180.000,B 0.000,C 180.000} C_DIS
LIN {X 90.282,Y 110.410,Z 68.000,A 180.000,B 0.000,C 180.000} C_DIS
LIN {X 90.414,Y 110.483,Z 68.000,A 180.000,B 0.000,C 180.000} C_DIS
LIN {X 90.997,Y 110.784,Z 68.000,A 180.000,B 0.000,C 180.000} C_DIS
LIN {X 91.111,Y 110.841,Z 68.000,A 180.000,B 0.000,C 180.000} C_DIS
LIN {X 91.176,Y 110.870,Z 68.000,A 180.000,B 0.000,C 180.000} C_DIS
LIN {X 91.712,Y 111.110,Z 68.000,A 180.000,B 0.000,C 180.000} C_DIS
LIN {X 91.891,Y 111.187,Z 68.000,A 180.000,B 0.000,C 180.000} C_DIS
LIN {X 91.921,Y 111.198,Z 68.000,A 180.000,B 0.000,C 180.000} C_DIS
LIN {X 92.427,Y 111.391,Z 68.000,A 180.000,B 0.000,C 180.000} C_DIS
LIN {X 92.606,Y 111.459,Z 68.000,A 180.000,B 0.000,C 180.000} C_DIS
LIN {X 92.785,Y 111.517,Z 68.000,A 180.000,B 0.000,C 180.000} C_DIS
LIN {X 93.321,Y 111.688,Z 68.000,A 180.000,B 0.000,C 180.000} C_DIS
LIN {X 93.482,Y 111.734,Z 68.000,A 180.000,B 0.000,C 180.000} C_DIS
LIN {X 94.036,Y 111.878,Z 68.000,A 180.000,B 0.000,C 180.000} C_DIS
LIN {X 94.176,Y 111.913,Z 68.000,A 180.000,B 0.000,C 180.000} C_DIS
LIN {X 94.215,Y 111.922,Z 68.000,A 180.000,B 0.000,C 180.000} C_DIS
LIN {X 94.394,Y 111.959,Z 68.000,A 180.000,B 0.000,C 180.000} C_DIS
LIN {X 94.930,Y 112.065,Z 68.000,A 180.000,B 0.000,C 180.000} C_DIS
LIN {X 95.080,Y 112.092,Z 68.000,A 180.000,B 0.000,C 180.000} C_DIS
LIN {X 95.109,Y 112.096,Z 68.000,A 180.000,B 0.000,C 180.000} C_DIS
LIN {X 95.645,Y 112.172,Z 68.000,A 180.000,B 0.000,C 180.000} C_DIS
LIN {X 95.824,Y 112.196,Z 68.000,A 180.000,B 0.000,C 180.000} C_DIS
LIN {X 96.003,Y 112.213,Z 68.000,A 180.000,B 0.000,C 180.000} C_DIS
LIN {X 96.539,Y 112.258,Z 68.000,A 180.000,B 0.000,C 180.000} C_DIS
LIN {X 96.718,Y 112.271,Z 68.000,A 180.000,B 0.000,C 180.000} C_DIS
LIN {X 96.719,Y 112.271,Z 68.000,A 180.000,B 0.000,C 180.000} C_DIS
LIN {X 96.897,Y 112.276,Z 68.000,A 180.000,B 0.000,C 180.000} C_DIS
LIN {X 97.433,Y 112.291,Z 68.000,A 180.000,B 0.000,C 180.000} C_DIS
LIN {X 97.612,Y 112.290,Z 68.000,A 180.000,B 0.000,C 180.000} C_DIS
LIN {X 98.148,Y 112.275,Z 68.000,A 180.000,B 0.000,C 180.000} C_DIS
LIN {X 98.281,Y 112.271,Z 68.000,A 180.000,B 0.000,C 180.000} C_DIS
LIN {X 98.327,Y 112.269,Z 68.000,A 180.000,B 0.000,C 180.000} C_DIS
LIN {X 98.505,Y 112.255,Z 68.000,A 180.000,B 0.000,C 180.000} C_DIS
LIN {X 99.042,Y 112.209,Z 68.000,A 180.000,B 0.000,C 180.000} C_DIS
LIN {X 99.221,Y 112.191,Z 68.000,A 180.000,B 0.000,C 180.000} C_DIS
LIN {X 99.757,Y 112.115,Z 68.000,A 180.000,B 0.000,C 180.000} C_DIS
LIN {X 99.920,Y 112.092,Z 68.000,A 180.000,B 0.000,C 180.000} C_DIS
LIN {X 99.936,Y 112.090,Z 68.000,A 180.000,B 0.000,C 180.000} C_DIS
LIN {X 100.114,Y 112.057,Z 68.000,A 180.000,B 0.000,C 180.000} C_DIS
LIN {X 100.651,Y 111.950,Z 68.000,A 180.000,B 0.000,C 180.000} C_DIS
LIN {X 100.824,Y 111.913,Z 68.000,A 180.000,B 0.000,C 180.000} C_DIS
LIN {X 100.829,Y 111.912,Z 68.000,A 180.000,B 0.000,C 180.000} C_DIS
LIN {X 101.008,Y 111.866,Z 68.000,A 180.000,B 0.000,C 180.000} C_DIS
LIN {X 101.518,Y 111.734,Z 68.000,A 180.000,B 0.000,C 180.000} C_DIS
LIN {X 101.545,Y 111.728,Z 68.000,A 180.000,B 0.000,C 180.000} C_DIS
LIN {X 101.723,Y 111.674,Z 68.000,A 180.000,B 0.000,C 180.000} C_DIS
LIN {X 102.260,Y 111.503,Z 68.000,A 180.000,B 0.000,C 180.000} C_DIS
LIN {X 102.438,Y 111.443,Z 68.000,A 180.000,B 0.000,C 180.000} C_DIS
LIN {X 102.617,Y 111.374,Z 68.000,A 180.000,B 0.000,C 180.000} C_DIS
LIN {X 103.079,Y 111.198,Z 68.000,A 180.000,B 0.000,C 180.000} C_DIS
LIN {X 103.153,Y 111.169,Z 68.000,A 180.000,B 0.000,C 180.000} C_DIS
LIN {X 103.332,Y 111.090,Z 68.000,A 180.000,B 0.000,C 180.000} C_DIS
LIN {X 103.690,Y 110.930,Z 68.000,A 180.000,B 0.000,C 180.000} C_DIS
LIN {X 103.869,Y 110.850,Z 68.000,A 180.000,B 0.000,C 180.000} C_DIS
LIN {X 103.889,Y 110.841,Z 68.000,A 180.000,B 0.000,C 180.000} C_DIS
LIN {X 104.047,Y 110.761,Z 68.000,A 180.000,B 0.000,C 180.000} C_DIS
LIN {X 104.586,Y 110.483,Z 68.000,A 180.000,B 0.000,C 180.000} C_DIS
